C09140=1217.409,7.610,-42.513,-179.514,5.457,148.808
C09141=1217.414,7.361,-42.498,-179.516,5.457,148.808
C09142=1217.419,7.111,-42.484,-179.519,5.456,148.809
C09143=1217.424,6.862,-42.470,-179.521,5.456,148.810
C09144=1217.430,6.611,-42.455,-179.524,5.455,148.810
C09145=1217.434,6.362,-42.440,-179.527,5.455,148.811
C09146=1217.439,6.113,-42.426,-179.529,5.455,148.812
C09147=1217.444,5.863,-42.411,-179.531,5.454,148.812
C09148=1217.450,5.614,-42.397,-179.534,5.454,148.813
C09149=1217.454,5.365,-42.382,-179.537,5.453,148.814
C09150=1217.459,5.115,-42.368,-179.539,5.453,148.814
C09151=1217.464,4.865,-42.354,-179.541,5.453,148.815
C09152=1217.469,4.616,-42.340,-179.544,5.453,148.816
C09153=1217.475,4.366,-42.324,-179.547,5.452,148.817
C09154=1217.480,4.117,-42.310,-179.549,5.452,148.817
C09155=1217.484,3.867,-42.295,-179.552,5.451,148.818
C09156=1217.490,3.598,-42.280,-179.555,5.451,148.819
C09157=1217.496,3.329,-42.265,-179.557,5.450,148.819
C09158=1217.501,3.061,-42.249,-179.559,5.450,148.820
C09159=1217.506,2.791,-42.234,-179.562,5.450,148.821
C09160=1217.511,2.542,-42.219,-179.565,5.449,148.821
C09161=1217.516,2.292,-42.205,-179.567,5.449,148.822
C09162=1217.521,2.043,-42.191,-179.570,5.448,148.823
C09163=1217.526,1.793,-42.176,-179.573,5.448,148.823
C09164=1217.532,1.544,-42.162,-179.575,5.448,148.824
C09165=1217.537,1.294,-42.148,-179.577,5.448,148.825
C09166=1217.542,1.044,-42.134,-179.580,5.447,148.825
C09167=1217.547,0.795,-42.119,-179.583,5.446,148.826
C09168=1217.552,0.545,-42.105,-179.585,5.446,148.827
C09169=1217.557,0.296,-42.091,-179.587,5.446,148.828
C09170=1217.562,0.046,-42.077,-179.589,5.445,148.828
C09171=1217.567,-0.203,-42.062,-179.592,5.445,148.829
C09172=1217.572,-0.453,-42.048,-179.595,5.444,148.829
C09173=1217.577,-0.702,-42.033,-179.597,5.445,148.830
C09174=1217.582,-0.951,-42.019,-179.600,5.444,148.831
C09175=1217.587,-1.201,-42.005,-179.602,5.444,148.831
C09176=1217.592,-1.451,-41.991,-179.605,5.443,148.832
C09177=1217.597,-1.700,-41.977,-179.608,5.443,148.833
C09178=1217.602,-1.950,-41.963,-179.610,5.443,148.833
C09179=1217.607,-2.199,-41.949,-179.612,5.442,148.834
C09180=1217.612,-2.449,-41.935,-179.615,5.442,148.835
C09181=1217.617,-2.698,-41.920,-179.618,5.441,148.836
C09182=1217.622,-2.948,-41.906,-179.620,5.442,148.836
C09183=1217.627,-3.198,-41.892,-179.622,5.441,148.837
C09184=1217.633,-3.447,-41.879,-179.625,5.441,148.838
C09185=1217.638,-3.697,-41.864,-179.628,5.440,148.838
C09186=1217.643,-3.947,-41.850,-179.629,5.440,148.839
C09187=1217.648,-4.197,-41.836,-179.632,5.440,148.839
C09188=1217.653,-4.446,-41.822,-179.634,5.439,148.840
C09189=1217.657,-4.695,-41.808,-179.637,5.439,148.841
C09190=1217.662,-4.945,-41.794,-179.640,5.438,148.842
C09191=1217.667,-5.194,-41.780,-179.642,5.438,148.842
C09192=1217.673,-5.443,-41.766,-179.645,5.438,148.843
C09193=1217.678,-5.693,-41.751,-179.647,5.437,148.844
C09194=1217.683,-5.943,-41.738,-179.650,5.437,148.844
C09195=1217.689,-6.192,-41.724,-179.652,5.437,148.845
C09196=1217.694,-6.442,-41.710,-179.655,5.437,148.846
C09197=1217.698,-6.692,-41.696,-179.657,5.436,148.846
C09198=1217.703,-6.941,-41.682,-179.660,5.436,148.847
C09199=1217.708,-7.190,-41.668,-179.662,5.436,148.848
C09200=1217.713,-7.440,-41.654,-179.665,5.435,148.848
C09201=1217.719,-7.690,-41.640,-179.667,5.435,148.849
C09202=1217.723,-7.939,-41.627,-179.670,5.434,148.850
C09203=1217.728,-8.189,-41.612,-179.672,5.435,148.851
C09204=1217.733,-8.438,-41.598,-179.674,5.434,148.851
C09205=1217.738,-8.688,-41.584,-179.677,5.433,148.852
C09206=1217.744,-8.938,-41.571,-179.679,5.433,148.852
C09207=1217.748,-9.187,-41.557,-179.682,5.433,148.853
C09208=1217.753,-9.437,-41.543,-179.684,5.433,148.854
C09209=1217.759,-9.686,-41.529,-179.687,5.432,148.854
C09210=1217.764,-9.936,-41.515,-179.689,5.432,148.855
C09211=1217.769,-10.186,-41.501,-179.692,5.432,148.856
C09212=1217.774,-10.435,-41.488,-179.694,5.431,148.857
C09213=1217.779,-10.684,-41.473,-179.697,5.431,148.857
C09214=1217.784,-10.935,-41.460,-179.700,5.430,148.858
C09215=1217.790,-11.184,-41.446,-179.702,5.431,148.859
C09216=1217.794,-11.433,-41.432,-179.704,5.430,148.859
C09217=1217.800,-11.683,-41.419,-179.707,5.430,148.860
C09218=1217.805,-11.932,-41.405,-179.710,5.429,148.861
C09219=1217.809,-12.182,-41.391,-179.712,5.430,148.861
C09220=1217.815,-12.431,-41.378,-179.714,5.429,148.862
C09221=1217.820,-12.681,-41.364,-179.717,5.429,148.863
C09222=1217.825,-12.931,-41.349,-179.720,5.428,148.863
C09223=1217.830,-13.180,-41.337,-179.722,5.428,148.864
C09224=1217.835,-13.430,-41.322,-179.724,5.427,148.865
C09225=1217.840,-13.680,-41.308,-179.727,5.427,148.865
C09226=1217.845,-13.929,-41.296,-179.729,5.427,148.866
C09227=1217.850,-14.179,-41.281,-179.731,5.427,148.867
C09228=1217.855,-14.428,-41.267,-179.734,5.426,148.867
C09229=1217.860,-14.678,-41.254,-179.737,5.426,148.868
C09230=1217.865,-14.927,-41.240,-179.739,5.426,148.869
C09231=1217.871,-15.177,-41.227,-179.741,5.426,148.869
C09232=1217.875,-15.426,-41.213,-179.744,5.425,148.870
C09233=1217.881,-15.676,-41.200,-179.747,5.425,148.871
C09234=1217.886,-15.926,-41.186,-179.749,5.425,148.872
C09235=1217.890,-16.174,-41.172,-179.751,5.424,148.872
C09236=1217.896,-16.425,-41.159,-179.754,5.424,148.873
C09237=1217.901,-16.674,-41.145,-179.756,5.424,148.874
C09238=1217.906,-16.924,-41.132,-179.759,5.424,148.874
C09239=1217.911,-17.174,-41.118,-179.761,5.423,148.875
C09240=1217.916,-17.423,-41.105,-179.764,5.423,148.876
C09241=1217.921,-17.673,-41.091,-179.766,5.423,148.876
C09242=1217.927,-17.922,-41.078,-179.769,5.423,148.877
C09243=1217.931,-18.172,-41.064,-179.771,5.422,148.878
C09244=1217.937,-18.421,-41.051,-179.774,5.422,148.878
C09245=1217.941,-18.671,-41.037,-179.776,5.422,148.879
C09246=1217.946,-18.921,-41.023,-179.778,5.421,148.880
C09247=1217.952,-19.170,-41.010,-179.781,5.420,148.880
C09248=1217.956,-19.420,-40.997,-179.783,5.421,148.881
C09249=1217.962,-19.669,-40.983,-179.786,5.420,148.882
C09250=1217.966,-19.919,-40.970,-179.788,5.420,148.882
C09251=1217.972,-20.169,-40.957,-179.791,5.420,148.883
C09252=1217.977,-20.418,-40.943,-179.793,5.420,148.884
C09253=1217.982,-20.668,-40.930,-179.796,5.419,148.884
C09254=1217.987,-20.917,-40.915,-179.798,5.419,148.885
C09255=1217.992,-21.167,-40.903,-179.801,5.419,148.886
C09256=1217.998,-21.417,-40.889,-179.803,5.418,148.887
C09257=1218.003,-21.666,-40.876,-179.806,5.418,148.887
C09258=1218.008,-21.916,-40.862,-179.808,5.418,148.888
C09259=1218.013,-22.165,-40.849,-179.811,5.418,148.889
C09260=1218.018,-22.435,-40.835,-179.813,5.417,148.889
C09261=1218.023,-22.704,-40.820,-179.816,5.417,148.890
C09262=1218.029,-22.973,-40.806,-179.819,5.416,148.891
C09263=1218.035,-23.243,-40.791,-179.821,5.417,148.892
C09264=1218.039,-23.493,-40.778,-179.824,5.417,148.892
C09265=1218.045,-23.742,-40.765,-179.827,5.416,148.893
C09266=1218.049,-23.992,-40.752,-179.829,5.416,148.894
C09267=1218.055,-24.241,-40.738,-179.831,5.416,148.894
C09268=1218.060,-24.491,-40.726,-179.833,5.415,148.895
C09269=1218.065,-24.740,-40.712,-179.836,5.414,148.896
C09270=1218.070,-24.990,-40.699,-179.838,5.415,148.896
C09271=1218.075,-25.240,-40.686,-179.841,5.414,148.897
C09272=1218.081,-25.489,-40.672,-179.843,5.414,148.898
C09273=1218.085,-25.739,-40.659,-179.846,5.414,148.898
C09274=1218.091,-25.988,-40.646,-179.848,5.414,148.899
C09275=1218.095,-26.238,-40.633,-179.851,5.413,148.900
C09276=1218.101,-26.487,-40.619,-179.853,5.413,148.901
C09277=1218.106,-26.737,-40.606,-179.856,5.413,148.901
C09278=1218.111,-26.987,-40.593,-179.858,5.412,148.902
C09279=1218.117,-27.236,-40.580,-179.860,5.413,148.903
C09280=1218.121,-27.486,-40.567,-179.863,5.412,148.903
C09281=1218.127,-27.735,-40.553,-179.866,5.412,148.904
C09282=1218.131,-27.985,-40.540,-179.868,5.411,148.905
C09283=1218.136,-28.235,-40.528,-179.870,5.412,148.905
C09284=1218.142,-28.484,-40.515,-179.873,5.411,148.906
C09285=1218.147,-28.734,-40.502,-179.876,5.411,148.907
C09286=1218.151,-28.983,-40.488,-179.878,5.411,148.907
C09287=1218.157,-29.233,-40.475,-179.880,5.411,148.908
C09288=1218.162,-29.483,-40.462,-179.883,5.410,148.909
C09289=1218.167,-29.732,-40.450,-179.885,5.410,148.910
C09290=1218.172,-29.982,-40.436,-179.888,5.410,148.910
C09291=1218.177,-30.232,-40.423,-179.891,5.409,148.911
C09292=1218.182,-30.482,-40.410,-179.893,5.410,148.912
C09293=1218.187,-30.731,-40.397,-179.895,5.409,148.912
C09294=1218.193,-30.980,-40.384,-179.897,5.408,148.913
C09295=1218.197,-31.230,-40.371,-179.900,5.409,148.914
C09296=1218.203,-31.480,-40.358,-179.902,5.408,148.914
C09297=1218.208,-31.729,-40.345,-179.905,5.408,148.915
C09298=1218.213,-31.979,-40.332,-179.907,5.408,148.916
C09299=1218.218,-32.229,-40.319,-179.910,5.408,148.916
C09300=1218.224,-32.478,-40.306,-179.912,5.407,148.917
C09301=1218.228,-32.728,-40.293,-179.914,5.407,148.918
C09302=1218.233,-32.977,-40.281,-179.917,5.407,148.918
C09303=1218.239,-33.227,-40.268,-179.920,5.406,148.919
C09304=1218.244,-33.477,-40.255,-179.922,5.407,148.920
C09305=1218.249,-33.726,-40.242,-179.924,5.406,148.921
C09306=1218.255,-33.976,-40.229,-179.927,5.406,148.921
C09307=1218.259,-34.226,-40.216,-179.929,5.406,148.922
C09308=1218.264,-34.475,-40.203,-179.932,5.406,148.923
C09309=1218.269,-34.724,-40.191,-179.934,5.405,148.923
C09310=1218.275,-34.975,-40.177,-179.937,5.405,148.924
C09311=1218.280,-35.224,-40.165,-179.939,5.405,148.925
C09312=1218.285,-35.473,-40.152,-179.942,5.404,148.925
C09313=1218.289,-35.723,-40.139,-179.944,5.405,148.926
C09314=1218.295,-35.973,-40.126,-179.947,5.404,148.927
C09315=1218.300,-36.222,-40.113,-179.949,5.404,148.928
C09316=1218.306,-36.472,-40.101,-179.951,5.404,148.928
C09317=1218.310,-36.722,-40.088,-179.954,5.404,148.929
C09318=1218.315,-36.971,-40.075,-179.957,5.403,148.930
C09319=1218.320,-37.220,-40.062,-179.958,5.403,148.930
C09320=1218.326,-37.471,-40.049,-179.961,5.403,148.931
C09321=1218.331,-37.720,-40.036,-179.963,5.403,148.931
C09322=1218.336,-37.969,-40.024,-179.966,5.403,148.932
C09323=1218.341,-38.219,-40.012,-179.968,5.402,148.933
C09324=1218.346,-38.469,-39.999,-179.970,5.402,148.934
C09325=1218.351,-38.719,-39.986,-179.973,5.402,148.934
C09326=1218.357,-38.968,-39.973,-179.976,5.401,148.935
C09327=1218.362,-39.218,-39.960,-179.978,5.402,148.936
C09328=1218.366,-39.468,-39.947,-179.981,5.401,148.936
C09329=1218.371,-39.717,-39.935,-179.983,5.401,148.937
C09330=1218.377,-39.967,-39.923,-179.985,5.401,148.938
C09331=1218.382,-40.216,-39.910,-179.988,5.401,148.938
C09332=1218.387,-40.466,-39.897,-179.991,5.400,148.939
C09333=1218.392,-40.716,-39.884,-179.993,5.400,148.940
C09334=1218.398,-40.965,-39.872,-179.995,5.400,148.941
C09335=1218.403,-41.214,-39.859,-179.997,5.400,148.941
C09336=1218.408,-41.464,-39.847,180.000,5.400,148.942
C09337=1218.413,-41.714,-39.834,179.997,5.399,148.943
C09338=1218.418,-41.964,-39.822,179.995,5.400,148.943
C09339=1218.423,-42.213,-39.809,179.992,5.399,148.944
C09340=1218.428,-42.463,-39.797,179.990,5.399,148.945
C09341=1218.433,-42.713,-39.784,179.988,5.399,148.945
C09342=1218.438,-42.962,-39.771,179.985,5.399,148.946
C09343=1218.443,-43.212,-39.759,179.982,5.398,148.947
C09344=1218.449,-43.462,-39.747,179.981,5.398,148.947
C09345=1218.454,-43.711,-39.734,179.978,5.398,148.948
C09346=1218.458,-43.961,-39.721,179.976,5.398,148.949
C09347=1218.464,-44.211,-39.708,179.973,5.397,148.949
C09348=1218.469,-44.460,-39.696,179.971,5.397,148.950
C09349=1218.475,-44.710,-39.684,179.969,5.397,148.951
C09350=1218.480,-44.959,-39.671,179.966,5.397,148.952
C09351=1218.485,-45.209,-39.659,179.963,5.396,148.952
C09352=1218.490,-45.459,-39.646,179.961,5.397,148.953
C09353=1218.495,-45.708,-39.634,179.959,5.396,148.954
C09354=1218.500,-45.958,-39.622,179.957,5.397,148.954
C09355=1218.505,-46.208,-39.609,179.954,5.396,148.955
C09356=1218.510,-46.457,-39.597,179.951,5.396,148.956
C09357=1218.516,-46.707,-39.585,179.949,5.396,148.956
C09358=1218.521,-46.956,-39.572,179.946,5.395,148.957
C09359=1218.526,-47.206,-39.559,179.944,5.395,148.958
C09360=1218.531,-47.456,-39.547,179.942,5.395,148.959
C09361=1218.536,-47.705,-39.535,179.939,5.395,148.959
C09362=1218.542,-47.955,-39.523,179.937,5.395,148.960
C09363=1218.546,-48.204,-39.511,179.934,5.395,148.961
C09364=1218.552,-48.475,-39.497,179.932,5.394,148.961
C09365=1218.558,-48.744,-39.484,179.929,5.394,148.962
C09366=1218.563,-49.014,-39.471,179.927,5.394,148.963
C09367=1218.568,-49.284,-39.457,179.924,5.394,148.964
C09368=1218.573,-49.534,-39.445,179.922,5.393,148.964
C09369=1218.578,-49.783,-39.433,179.919,5.394,148.965
C09370=1218.584,-50.033,-39.420,179.917,5.393,148.966
C09371=1218.589,-50.283,-39.408,179.915,5.393,148.966
C09372=1218.594,-50.532,-39.396,179.912,5.393,148.967
C09373=1218.600,-50.782,-39.384,179.909,5.392,148.968
C09374=1218.605,-51.031,-39.371,179.907,5.393,148.968
C09375=1218.610,-51.281,-39.359,179.905,5.392,148.969
C09376=1218.615,-51.531,-39.346,179.902,5.392,148.970
C09377=1218.619,-51.781,-39.335,179.900,5.392,148.971
C09378=1218.624,-52.030,-39.322,179.897,5.392,148.971
C09379=1218.630,-52.280,-39.311,179.895,5.392,148.972
C09380=1218.635,-52.529,-39.298,179.892,5.392,148.973
C09381=1218.640,-52.779,-39.286,179.890,5.391,148.973
C09382=1218.646,-53.029,-39.274,179.888,5.391,148.974
C09383=1218.651,-53.279,-39.262,179.885,5.391,148.975
C09384=1218.656,-53.528,-39.250,179.883,5.391,148.975
C09385=1218.661,-53.778,-39.238,179.880,5.391,148.976
C09386=1218.666,-54.027,-39.226,179.878,5.390,148.977
C09387=1218.671,-54.277,-39.213,179.876,5.391,148.978
C09388=1218.677,-54.527,-39.201,179.873,5.390,148.978
C09389=1218.682,-54.776,-39.189,179.871,5.390,148.979
C09390=1218.687,-55.026,-39.177,179.869,5.390,148.979
C09391=1218.692,-55.276,-39.166,179.866,5.389,148.980
C09392=1218.697,-55.526,-39.153,179.864,5.390,148.981
C09393=1218.702,-55.776,-39.141,179.861,5.389,148.982
C09394=1218.707,-56.026,-39.129,179.859,5.390,148.982
C09395=1218.712,-56.275,-39.117,179.856,5.389,148.983
C09396=1218.717,-56.524,-39.105,179.854,5.389,148.984
C09397=1218.722,-56.774,-39.092,179.852,5.389,148.984
C09398=1218.728,-57.024,-39.080,179.849,5.388,148.985
C09399=1218.732,-57.273,-39.069,179.847,5.389,148.986
C09400=1218.738,-57.523,-39.057,179.844,5.388,148.987
C09401=1218.743,-57.773,-39.045,179.842,5.389,148.987
C09402=1218.748,-58.023,-39.033,179.839,5.388,148.988
C09403=1218.753,-58.272,-39.021,179.837,5.388,148.989
C09404=1218.758,-58.521,-39.009,179.835,5.388,148.989
C09405=1218.764,-58.771,-38.997,179.832,5.388,148.990
C09406=1218.769,-59.021,-38.985,179.830,5.388,148.991
C09407=1218.773,-59.270,-38.973,179.827,5.388,148.991
C09408=1218.779,-59.520,-38.961,179.825,5.387,148.992
C09409=1218.784,-59.770,-38.949,179.823,5.387,148.993
C09410=1218.790,-60.019,-38.938,179.820,5.387,148.993
C09411=1218.795,-60.268,-38.926,179.818,5.387,148.994
C09412=1218.800,-60.518,-38.914,179.816,5.386,148.995
C09413=1218.806,-60.768,-38.902,179.813,5.386,148.995
C09414=1218.810,-61.018,-38.891,179.811,5.386,148.996
C09415=1218.815,-61.267,-38.878,179.808,5.386,148.997
C09416=1218.821,-61.517,-38.866,179.806,5.386,148.998
C09417=1218.826,-61.767,-38.855,179.803,5.386,148.998
C09418=1218.831,-62.017,-38.843,179.801,5.386,148.999
C09419=1218.836,-62.267,-38.831,179.799,5.386,149.000
C09420=1218.841,-62.516,-38.819,179.796,5.385,149.000
C09421=1218.846,-62.766,-38.807,179.794,5.385,149.001
C09422=1218.852,-63.016,-38.795,179.791,5.385,149.002
C09423=1218.856,-63.265,-38.784,179.789,5.385,149.002
C09424=1218.862,-63.515,-38.772,179.787,5.385,149.003
C09425=1218.866,-63.765,-38.761,179.784,5.385,149.004
C09426=1218.872,-64.013,-38.749,179.782,5.384,149.004
C09427=1218.878,-64.263,-38.737,179.780,5.384,149.005
C09428=1218.882,-64.513,-38.726,179.778,5.384,149.006
C09429=1218.888,-64.763,-38.714,179.775,5.384,149.007
C09430=1218.893,-65.013,-38.702,179.773,5.384,149.007
C09431=1218.898,-65.262,-38.691,179.770,5.384,149.008
C09432=1218.903,-65.512,-38.679,179.768,5.384,149.009
C09433=1218.908,-65.762,-38.667,179.765,5.384,149.009
C09434=1218.913,-66.012,-38.655,179.763,5.383,149.010
C09435=1218.918,-66.261,-38.643,179.761,5.384,149.011
C09436=1218.924,-66.510,-38.632,179.758,5.383,149.011
C09437=1218.929,-66.760,-38.620,179.756,5.383,149.012
C09438=1218.934,-67.010,-38.609,179.753,5.383,149.013
C09439=1218.939,-67.260,-38.597,179.751,5.383,149.014
C09440=1218.944,-67.509,-38.586,179.748,5.383,149.014
C09441=1218.949,-67.759,-38.574,179.746,5.382,149.015
C09442=1218.954,-68.009,-38.562,179.744,5.382,149.015
C09443=1218.960,-68.258,-38.551,179.741,5.382,149.016
C09444=1218.966,-68.508,-38.539,179.739,5.382,149.017
C09445=1218.970,-68.758,-38.528,179.737,5.382,149.018
C09446=1218.976,-69.008,-38.516,179.735,5.382,149.018
C09447=1218.980,-69.257,-38.505,179.732,5.382,149.019
C09448=1218.986,-69.507,-38.493,179.730,5.382,149.020
C09449=1218.991,-69.756,-38.482,179.727,5.382,149.020
C09450=1218.997,-70.006,-38.470,179.724,5.381,149.021
C09451=1219.001,-70.256,-38.459,179.722,5.381,149.022
C09452=1219.007,-70.506,-38.447,179.720,5.381,149.023
C09453=1219.011,-70.755,-38.435,179.718,5.381,149.023
C09454=1219.017,-71.005,-38.423,179.715,5.381,149.024
C09455=1219.022,-71.254,-38.413,179.713,5.381,149.025
C09456=1219.028,-71.504,-38.401,179.710,5.381,149.025
C09457=1219.033,-71.754,-38.390,179.709,5.381,149.026
C09458=1219.038,-72.004,-38.378,179.706,5.380,149.027
C09459=1219.043,-72.254,-38.367,179.703,5.380,149.027
C09460=1219.049,-72.503,-38.355,179.701,5.380,149.028
C09461=1219.053,-72.753,-38.344,179.699,5.380,149.029
C09462=1219.058,-73.002,-38.333,179.696,5.380,149.029
C09463=1219.064,-73.252,-38.321,179.694,5.380,149.030
C09464=1219.069,-73.501,-38.310,179.692,5.380,149.031
C09465=1219.074,-73.751,-38.298,179.689,5.380,149.032
C09466=1219.079,-74.001,-38.288,179.687,5.380,149.032
C09467=1219.085,-74.251,-38.276,179.684,5.379,149.033
C09468=1219.091,-74.521,-38.263,179.682,5.379,149.034
C09469=1219.095,-74.792,-38.251,179.680,5.379,149.034
C09470=1219.101,-75.063,-38.239,179.677,5.379,149.035
C09471=1219.107,-75.332,-38.227,179.674,5.379,149.036
C09472=1219.112,-75.583,-38.216,179.672,5.379,149.036
C09473=1219.117,-75.832,-38.204,179.669,5.378,149.037
C09474=1219.122,-76.082,-38.193,179.667,5.379,149.038
C09475=1219.128,-76.331,-38.181,179.665,5.378,149.039
C09476=1219.133,-76.581,-38.170,179.663,5.379,149.039
C09477=1219.138,-76.831,-38.159,179.660,5.378,149.040
C09478=1219.144,-77.080,-38.148,179.658,5.379,149.041
C09479=1219.149,-77.330,-38.137,179.655,5.378,149.041
C09480=1219.154,-77.580,-38.125,179.652,5.378,149.042
C09481=1219.159,-77.830,-38.114,179.650,5.378,149.043
C09482=1219.164,-78.079,-38.103,179.648,5.377,149.043
C09483=1219.170,-78.329,-38.091,179.646,5.378,149.044
C09484=1219.174,-78.579,-38.080,179.643,5.377,149.045
C09485=1219.179,-78.829,-38.069,179.641,5.377,149.045
C09486=1219.185,-79.078,-38.058,179.639,5.377,149.046
C09487=1219.190,-79.328,-38.047,179.637,5.377,149.047
C09488=1219.195,-79.578,-38.036,179.634,5.377,149.048
C09489=1219.200,-79.827,-38.025,179.632,5.377,149.048
C09490=1219.206,-80.077,-38.013,179.629,5.377,149.049
C09491=1219.211,-80.327,-38.002,179.627,5.377,149.050
C09492=1219.216,-80.576,-37.992,179.624,5.377,149.050
C09493=1219.222,-80.826,-37.980,179.622,5.377,149.051
C09494=1219.226,-81.076,-37.969,179.620,5.376,149.052
C09495=1219.232,-81.325,-37.958,179.617,5.376,149.052
C09496=1219.237,-81.575,-37.947,179.615,5.376,149.053
C09497=1219.242,-81.825,-37.936,179.613,5.376,149.054
C09498=1219.248,-82.074,-37.925,179.611,5.376,149.054
C09499=1219.252,-82.324,-37.914,179.608,5.376,149.055
C09500=1219.258,-82.574,-37.903,179.606,5.376,149.056
C09501=1219.263,-82.823,-37.892,179.603,5.376,149.057
C09502=1219.268,-83.073,-37.880,179.601,5.376,149.057
C09503=1219.273,-83.323,-37.870,179.598,5.376,149.058
C09504=1219.278,-83.572,-37.859,179.596,5.376,149.059
C09505=1219.284,-83.823,-37.848,179.594,5.375,149.059
C09506=1219.289,-84.072,-37.836,179.592,5.375,149.060
C09507=1219.294,-84.321,-37.825,179.589,5.375,149.061
C09508=1219.299,-84.572,-37.815,179.587,5.375,149.061
C09509=1219.304,-84.821,-37.803,179.585,5.375,149.062
C09510=1219.310,-85.071,-37.793,179.583,5.375,149.063
C09511=1219.315,-85.321,-37.782,179.580,5.375,149.063
C09512=1219.320,-85.570,-37.771,179.578,5.375,149.064
C09513=1219.325,-85.820,-37.760,179.575,5.375,149.065
C09514=1219.331,-86.070,-37.749,179.572,5.374,149.066
C09515=1219.336,-86.319,-37.738,179.571,5.374,149.066
C09516=1219.341,-86.570,-37.727,179.568,5.374,149.067
C09517=1219.346,-86.819,-37.716,179.566,5.374,149.067
C09518=1219.351,-87.069,-37.706,179.563,5.374,149.068
C09519=1219.356,-87.318,-37.695,179.561,5.374,149.069
C09520=1219.362,-87.568,-37.684,179.559,5.374,149.070
C09521=1219.367,-87.818,-37.672,179.557,5.374,149.070
C09522=1219.372,-88.068,-37.662,179.554,5.374,149.071
C09523=1219.377,-88.317,-37.651,179.552,5.374,149.072
C09524=1219.382,-88.567,-37.640,179.549,5.373,149.072
C09525=1219.388,-88.816,-37.629,179.547,5.373,149.073
C09526=1219.393,-89.066,-37.619,179.545,5.373,149.074
C09527=1219.398,-89.315,-37.608,179.543,5.373,149.074
C09528=1219.404,-89.566,-37.597,179.540,5.373,149.075
C09529=1219.409,-89.816,-37.586,179.538,5.373,149.076
C09530=1219.414,-90.065,-37.575,179.535,5.373,149.076
C09531=1219.419,-90.315,-37.565,179.533,5.373,149.077
C09532=1219.424,-90.564,-37.554,179.531,5.373,149.078
C09533=1219.429,-90.814,-37.543,179.528,5.373,149.079
C09534=1219.435,-91.064,-37.533,179.526,5.372,149.079
C09535=1219.440,-91.314,-37.522,179.524,5.373,149.080
C09536=1219.445,-91.563,-37.512,179.521,5.372,149.081
C09537=1219.450,-91.813,-37.501,179.519,5.373,149.081
C09538=1219.455,-92.062,-37.490,179.517,5.372,149.082
C09539=1219.460,-92.313,-37.479,179.515,5.373,149.083
C09540=1219.466,-92.563,-37.468,179.512,5.372,149.083
C09541=1219.471,-92.812,-37.457,179.510,5.373,149.084
C09542=1219.476,-93.062,-37.447,179.508,5.372,149.085
C09543=1219.482,-93.311,-37.436,179.506,5.372,149.085
C09544=1219.487,-93.561,-37.425,179.503,5.372,149.086
C09545=1219.492,-93.811,-37.415,179.501,5.372,149.087
C09546=1219.497,-94.061,-37.404,179.498,5.372,149.087
C09547=1219.503,-94.310,-37.394,179.496,5.372,149.088
C09548=1219.508,-94.560,-37.383,179.493,5.371,149.089
C09549=1219.513,-94.810,-37.373,179.491,5.372,149.090
C09550=1219.518,-95.060,-37.361,179.489,5.371,149.090
C09551=1219.523,-95.309,-37.351,179.487,5.371,149.091
C09552=1219.528,-95.559,-37.341,179.484,5.371,149.091
C09553=1219.534,-95.809,-37.330,179.482,5.371,149.092
C09554=1219.539,-96.059,-37.319,179.480,5.371,149.093
C09555=1219.544,-96.308,-37.309,179.477,5.371,149.094
C09556=1219.550,-96.558,-37.299,179.475,5.371,149.094
C09557=1219.555,-96.808,-37.288,179.473,5.371,149.095
C09558=1219.560,-97.057,-37.277,179.471,5.370,149.096
C09559=1219.565,-97.307,-37.267,179.468,5.371,149.096
C09560=1219.571,-97.557,-37.257,179.466,5.370,149.097
C09561=1219.576,-97.807,-37.246,179.464,5.371,149.098
C09562=1219.581,-98.056,-37.236,179.461,5.370,149.098
C09563=1219.586,-98.306,-37.224,179.459,5.371,149.099
C09564=1219.591,-98.555,-37.215,179.456,5.370,149.100
C09565=1219.596,-98.806,-37.204,179.454,5.371,149.100
C09566=1219.602,-99.055,-37.194,179.452,5.370,149.101
C09567=1219.607,-99.305,-37.184,179.450,5.370,149.102
C09568=1219.612,-99.555,-37.173,179.447,5.370,149.102
C09569=1219.617,-99.804,-37.162,179.445,5.370,149.103
C09570=1219.622,-100.054,-37.152,179.442,5.370,149.104
C09571=1219.628,-100.304,-37.142,179.440,5.370,149.105
C09572=1219.633,-100.575,-37.131,179.438,5.370,149.105
C09573=1219.639,-100.846,-37.119,179.435,5.369,149.106
C09574=1219.645,-101.117,-37.108,179.433,5.370,149.107
C09575=1219.651,-101.388,-37.096,179.430,5.369,149.107
C09576=1219.656,-101.638,-37.086,179.428,5.369,149.108
C09577=1219.661,-101.888,-37.075,179.425,5.369,149.109
C09578=1219.666,-102.137,-37.066,179.423,5.369,149.110
C09579=1219.671,-102.387,-37.055,179.421,5.369,149.110
C09580=1219.677,-102.637,-37.045,179.419,5.369,149.111
C09581=1219.682,-102.886,-37.035,179.416,5.369,149.111
C09582=1219.687,-103.137,-37.024,179.414,5.369,149.112
C09583=1219.693,-103.386,-37.014,179.412,5.368,149.113
C09584=1219.698,-103.636,-37.003,179.410,5.369,149.114
C09585=1219.703,-103.886,-36.994,179.407,5.368,149.114
C09586=1219.708,-104.135,-36.984,179.405,5.369,149.115
C09587=1219.713,-104.385,-36.973,179.403,5.368,149.116
C09588=1219.719,-104.635,-36.963,179.401,5.368,149.116
C09589=1219.724,-104.885,-36.953,179.398,5.368,149.117
C09590=1219.729,-105.134,-36.943,179.396,5.368,149.118
C09591=1219.734,-105.384,-36.932,179.393,5.368,149.118
C09592=1219.739,-105.634,-36.922,179.391,5.368,149.119
C09593=1219.745,-105.884,-36.912,179.389,5.368,149.120
C09594=1219.751,-106.133,-36.902,179.387,5.368,149.120
C09595=1219.755,-106.383,-36.892,179.385,5.368,149.121
C09596=1219.760,-106.633,-36.881,179.382,5.368,149.122
C09597=1219.766,-106.882,-36.871,179.380,5.368,149.122
C09598=1219.771,-107.133,-36.861,179.377,5.368,149.123
C09599=1219.776,-107.382,-36.851,179.375,5.368,149.124
C09600=1219.781,-107.631,-36.841,179.373,5.367,149.124
C09601=1219.786,-107.882,-36.830,179.371,5.368,149.125
C09602=1219.792,-108.131,-36.820,179.368,5.367,149.126
C09603=1219.798,-108.381,-36.810,179.366,5.368,149.126
C09604=1219.802,-108.631,-36.800,179.363,5.367,149.127
C09605=1219.808,-108.880,-36.790,179.361,5.368,149.128
C09606=1219.813,-109.130,-36.779,179.359,5.367,149.128
C09607=1219.818,-109.380,-36.770,179.357,5.367,149.129
C09608=1219.823,-109.630,-36.760,179.354,5.367,149.130
C09609=1219.829,-109.879,-36.750,179.352,5.367,149.131
C09610=1219.834,-110.129,-36.739,179.350,5.367,149.131
C09611=1219.839,-110.379,-36.729,179.347,5.367,149.132
C09612=1219.844,-110.628,-36.719,179.345,5.366,149.132
C09613=1219.850,-110.878,-36.709,179.343,5.367,149.133
C09614=1219.854,-111.128,-36.699,179.341,5.367,149.134
C09615=1219.860,-111.378,-36.690,179.338,5.367,149.135
C09616=1219.866,-111.628,-36.679,179.336,5.367,149.135
C09617=1219.871,-111.877,-36.670,179.334,5.366,149.136
C09618=1219.876,-112.127,-36.659,179.332,5.367,149.136
C09619=1219.881,-112.377,-36.649,179.329,5.366,149.137
C09620=1219.886,-112.626,-36.640,179.327,5.366,149.138
C09621=1219.892,-112.876,-36.630,179.325,5.366,149.139
C09622=1219.897,-113.126,-36.619,179.322,5.366,149.139
C09623=1219.902,-113.375,-36.610,179.320,5.366,149.140
C09624=1219.907,-113.625,-36.599,179.318,5.366,149.141
C09625=1219.913,-113.875,-36.590,179.316,5.366,149.141
C09626=1219.918,-114.125,-36.580,179.313,5.366,149.142
C09627=1219.923,-114.375,-36.570,179.311,5.366,149.143
C09628=1219.929,-114.624,-36.560,179.309,5.366,149.143
C09629=1219.934,-114.874,-36.551,179.307,5.366,149.144
C09630=1219.939,-115.124,-36.540,179.304,5.366,149.145
C09631=1219.944,-115.374,-36.530,179.302,5.366,149.145
C09632=1219.949,-115.623,-36.520,179.300,5.365,149.146
C09633=1219.955,-115.873,-36.511,179.298,5.365,149.147
C09634=1219.960,-116.122,-36.501,179.295,5.365,149.147
C09635=1219.965,-116.373,-36.491,179.293,5.365,149.148
C09636=1219.971,-116.623,-36.481,179.291,5.365,149.149
C09637=1219.976,-116.872,-36.471,179.288,5.365,149.149
C09638=1219.981,-117.122,-36.461,179.286,5.365,149.150
C09639=1219.987,-117.371,-36.452,179.284,5.365,149.151
C09640=1219.992,-117.622,-36.442,179.281,5.365,149.151
C09641=1219.997,-117.871,-36.432,179.279,5.365,149.152
C09642=1220.002,-118.121,-36.423,179.277,5.365,149.153
C09643=1220.008,-118.371,-36.412,179.275,5.365,149.153
C09644=1220.013,-118.620,-36.403,179.273,5.365,149.154
C09645=1220.018,-118.871,-36.393,179.270,5.364,149.155
C09646=1220.023,-119.120,-36.383,179.268,5.365,149.155
C09647=1220.029,-119.370,-36.373,179.266,5.364,149.156
C09648=1220.034,-119.619,-36.364,179.264,5.364,149.157
C09649=1220.039,-119.869,-36.354,179.261,5.364,149.157
C09650=1220.044,-120.119,-36.345,179.259,5.364,149.158
C09651=1220.050,-120.369,-36.335,179.257,5.364,149.159
C09652=1220.054,-120.618,-36.325,179.254,5.364,149.159
C09653=1220.060,-120.868,-36.316,179.252,5.364,149.160
C09654=1220.065,-121.118,-36.306,179.250,5.364,149.161
C09655=1220.071,-121.368,-36.296,179.248,5.364,149.161
C09656=1220.076,-121.617,-36.287,179.245,5.364,149.162
C09657=1220.081,-121.868,-36.277,179.243,5.364,149.163
C09658=1220.086,-122.117,-36.267,179.241,5.364,149.163
C09659=1220.092,-122.367,-36.257,179.239,5.364,149.164
C09660=1220.097,-122.617,-36.248,179.236,5.363,149.165
C09661=1220.102,-122.866,-36.238,179.234,5.364,149.165
C09662=1220.108,-123.116,-36.229,179.232,5.363,149.166
C09663=1220.113,-123.365,-36.219,179.230,5.363,149.167
C09664=1220.118,-123.616,-36.210,179.227,5.363,149.167
C09665=1220.123,-123.865,-36.200,179.225,5.363,149.168
C09666=1220.129,-124.115,-36.191,179.223,5.364,149.169
C09667=1220.133,-124.365,-36.181,179.221,5.363,149.169
C09668=1220.139,-124.615,-36.171,179.219,5.363,149.170
C09669=1220.144,-124.864,-36.162,179.216,5.363,149.171
C09670=1220.150,-125.114,-36.152,179.214,5.363,149.171
C09671=1220.155,-125.363,-36.143,179.212,5.363,149.172
C09672=1220.160,-125.613,-36.134,179.210,5.363,149.173
C09673=1220.166,-125.863,-36.124,179.207,5.363,149.173
C09674=1220.170,-126.113,-36.114,179.205,5.363,149.174
C09675=1220.176,-126.364,-36.105,179.202,5.363,149.175
C09676=1219.755,-126.374,-36.142,179.198,5.366,149.177
C09677=1219.749,-126.123,-36.151,179.201,5.366,149.176
C09678=1219.744,-125.874,-36.161,179.203,5.366,149.175
C09679=1219.738,-125.624,-36.170,179.205,5.367,149.175
C09680=1219.734,-125.375,-36.180,179.207,5.366,149.174
C09681=1219.728,-125.125,-36.189,179.210,5.367,149.173
C09682=1219.723,-124.875,-36.199,179.212,5.366,149.173
C09683=1219.718,-124.626,-36.208,179.214,5.367,149.172
C09684=1219.712,-124.375,-36.217,179.216,5.367,149.171
C09685=1219.707,-124.126,-36.227,179.219,5.367,149.171
C09686=1219.702,-123.875,-36.237,179.221,5.367,149.170
C09687=1219.697,-123.626,-36.246,179.223,5.367,149.169
C09688=1219.691,-123.376,-36.255,179.226,5.367,149.169
C09689=1219.686,-123.127,-36.265,179.228,5.367,149.168
C09690=1219.681,-122.877,-36.275,179.230,5.367,149.167
C09691=1219.675,-122.627,-36.285,179.232,5.367,149.167
C09692=1219.670,-122.378,-36.294,179.235,5.367,149.166
C09693=1219.664,-122.128,-36.304,179.237,5.367,149.165
C09694=1219.660,-121.878,-36.314,179.239,5.367,149.165
C09695=1219.654,-121.628,-36.323,179.241,5.367,149.164
C09696=1219.649,-121.379,-36.333,179.244,5.368,149.163
C09697=1219.643,-121.128,-36.342,179.246,5.368,149.163
C09698=1219.639,-120.879,-36.352,179.248,5.367,149.162
C09699=1219.633,-120.629,-36.361,179.250,5.368,149.161
C09700=1219.628,-120.380,-36.371,179.253,5.367,149.161
C09701=1219.623,-120.130,-36.382,179.255,5.368,149.160
C09702=1219.618,-119.880,-36.390,179.257,5.368,149.159
C09703=1219.612,-119.630,-36.401,179.260,5.368,149.159
C09704=1219.607,-119.380,-36.410,179.262,5.368,149.158
C09705=1219.601,-119.131,-36.420,179.264,5.368,149.157
C09706=1219.596,-118.882,-36.429,179.266,5.368,149.157
C09707=1219.591,-118.631,-36.439,179.269,5.368,149.156
C09708=1219.586,-118.381,-36.449,179.271,5.368,149.155
C09709=1219.581,-118.132,-36.459,179.273,5.368,149.155
C09710=1219.575,-117.882,-36.468,179.275,5.368,149.154
C09711=1219.570,-117.632,-36.478,179.277,5.368,149.153
C09712=1219.565,-117.382,-36.489,179.280,5.369,149.153
C09713=1219.560,-117.132,-36.498,179.282,5.368,149.152
C09714=1219.554,-116.883,-36.508,179.285,5.369,149.151
C09715=1219.549,-116.634,-36.517,179.286,5.369,149.151
C09716=1219.543,-116.383,-36.527,179.289,5.369,149.150
C09717=1219.539,-116.133,-36.537,179.291,5.369,149.149
C09718=1219.533,-115.884,-36.547,179.294,5.369,149.149
C09719=1219.528,-115.634,-36.557,179.296,5.369,149.148
C09720=1219.523,-115.385,-36.566,179.298,5.369,149.147
C09721=1219.518,-115.134,-36.577,179.300,5.369,149.147
C09722=1219.512,-114.885,-36.587,179.302,5.369,149.146
C09723=1219.507,-114.635,-36.596,179.305,5.369,149.145
C09724=1219.501,-114.385,-36.606,179.307,5.369,149.145
C09725=1219.497,-114.136,-36.616,179.309,5.369,149.144
C09726=1219.492,-113.886,-36.626,179.311,5.369,149.143
C09727=1219.486,-113.636,-36.636,179.314,5.370,149.143
C09728=1219.481,-113.387,-36.645,179.316,5.369,149.142
C09729=1219.475,-113.137,-36.656,179.319,5.370,149.141
C09730=1219.470,-112.887,-36.666,179.321,5.369,149.141
C09731=1219.465,-112.637,-36.675,179.323,5.370,149.140
C09732=1219.459,-112.387,-36.685,179.325,5.370,149.139
C09733=1219.454,-112.138,-36.696,179.328,5.370,149.139
C09734=1219.450,-111.888,-36.706,179.330,5.370,149.138
C09735=1219.444,-111.638,-36.716,179.332,5.370,149.137
C09736=1219.438,-111.389,-36.726,179.334,5.370,149.137
C09737=1219.433,-111.139,-36.735,179.337,5.371,149.136
C09738=1219.428,-110.889,-36.745,179.339,5.370,149.135
C09739=1219.423,-110.639,-36.756,179.341,5.370,149.135
C09740=1219.418,-110.390,-36.765,179.343,5.370,149.134
C09741=1219.413,-110.140,-36.776,179.346,5.370,149.133
C09742=1219.407,-109.890,-36.786,179.348,5.371,149.133
C09743=1219.401,-109.640,-36.795,179.350,5.370,149.132
C09744=1219.397,-109.390,-36.805,179.353,5.371,149.131
C09745=1219.391,-109.140,-36.816,179.355,5.370,149.130
C09746=1219.386,-108.891,-36.826,179.357,5.371,149.130
C09747=1219.381,-108.642,-36.836,179.359,5.370,149.129
C09748=1219.376,-108.391,-36.846,179.362,5.371,149.129
C09749=1219.370,-108.142,-36.856,179.364,5.371,149.128
C09750=1219.365,-107.892,-36.866,179.366,5.371,149.127
C09751=1219.360,-107.642,-36.876,179.368,5.371,149.126
C09752=1219.355,-107.393,-36.887,179.371,5.371,149.126
C09753=1219.349,-107.143,-36.897,179.373,5.371,149.125
C09754=1219.344,-106.892,-36.907,179.375,5.372,149.125
C09755=1219.339,-106.643,-36.916,179.377,5.371,149.124
C09756=1219.333,-106.394,-36.927,179.380,5.372,149.123
C09757=1219.328,-106.143,-36.937,179.382,5.371,149.122
C09758=1219.323,-105.894,-36.947,179.385,5.372,149.122
C09759=1219.317,-105.644,-36.958,179.387,5.371,149.121
C09760=1219.313,-105.394,-36.968,179.389,5.371,149.120
C09761=1219.307,-105.145,-36.978,179.391,5.372,149.120
C09762=1219.302,-104.895,-36.988,179.393,5.371,149.119
C09763=1219.297,-104.645,-36.999,179.396,5.372,149.118
C09764=1219.291,-104.396,-37.009,179.398,5.372,149.118
C09765=1219.287,-104.146,-37.019,179.401,5.372,149.117
C09766=1219.281,-103.896,-37.029,179.402,5.372,149.116
C09767=1219.276,-103.647,-37.039,179.405,5.372,149.116
C09768=1219.271,-103.396,-37.050,179.407,5.372,149.115
C09769=1219.265,-103.147,-37.060,179.410,5.372,149.114
C09770=1219.260,-102.898,-37.071,179.412,5.372,149.114
C09771=1219.256,-102.648,-37.081,179.415,5.372,149.113
C09772=1219.250,-102.398,-37.091,179.417,5.372,149.112
C09773=1219.245,-102.148,-37.102,179.419,5.373,149.112
C09774=1219.239,-101.899,-37.112,179.421,5.373,149.111
C09775=1219.234,-101.649,-37.122,179.424,5.373,149.110
C09776=1219.229,-101.399,-37.133,179.426,5.373,149.110
C09777=1219.224,-101.127,-37.144,179.428,5.373,149.109
C09778=1219.217,-100.857,-37.155,179.431,5.373,149.108
C09779=1219.212,-100.586,-37.166,179.433,5.373,149.107
C09780=1219.206,-100.314,-37.178,179.436,5.374,149.107
C09781=1219.201,-100.065,-37.188,179.438,5.373,149.106
C09782=1219.196,-99.815,-37.198,179.441,5.374,149.105
C09783=1219.191,-99.565,-37.208,179.443,5.373,149.105
C09784=1219.185,-99.316,-37.219,179.445,5.374,149.104
C09785=1219.180,-99.065,-37.229,179.448,5.373,149.103
C09786=1219.175,-98.817,-37.240,179.450,5.374,149.102
C09787=1219.170,-98.566,-37.251,179.452,5.374,149.102
C09788=1219.164,-98.317,-37.261,179.454,5.374,149.101
C09789=1219.159,-98.067,-37.271,179.457,5.374,149.100
C09790=1219.154,-97.817,-37.282,179.459,5.374,149.100
C09791=1219.149,-97.567,-37.292,179.461,5.374,149.099
C09792=1219.143,-97.318,-37.303,179.464,5.374,149.098
C09793=1219.138,-97.068,-37.313,179.466,5.374,149.098
C09794=1219.133,-96.818,-37.324,179.468,5.375,149.097
C09795=1219.127,-96.568,-37.334,179.470,5.374,149.096
C09796=1219.123,-96.319,-37.345,179.473,5.375,149.096
C09797=1219.117,-96.069,-37.356,179.475,5.374,149.095
C09798=1219.112,-95.819,-37.366,179.478,5.375,149.094
C09799=1219.106,-95.570,-37.376,179.480,5.374,149.094
C09800=1219.102,-95.320,-37.388,179.483,5.375,149.093
C09801=1219.096,-95.070,-37.398,179.485,5.375,149.092
C09802=1219.091,-94.820,-37.408,179.487,5.375,149.092
C09803=1219.086,-94.571,-37.419,179.489,5.375,149.091
C09804=1219.081,-94.321,-37.430,179.492,5.375,149.090
C09805=1219.075,-94.071,-37.440,179.494,5.375,149.090
C09806=1219.070,-93.821,-37.451,179.496,5.375,149.089
C09807=1219.065,-93.572,-37.462,179.498,5.375,149.088
C09808=1219.060,-93.322,-37.472,179.501,5.376,149.087
C09809=1219.054,-93.072,-37.482,179.503,5.375,149.087
C09810=1219.049,-92.822,-37.493,179.505,5.376,149.086
C09811=1219.044,-92.573,-37.504,179.507,5.376,149.085
C09812=1219.039,-92.323,-37.514,179.510,5.376,149.085
C09813=1219.033,-92.073,-37.525,179.512,5.376,149.084
C09814=1219.029,-91.824,-37.536,179.515,5.376,149.083
C09815=1219.023,-91.574,-37.546,179.517,5.376,149.083
C09816=1219.018,-91.325,-37.557,179.520,5.376,149.082
C09817=1219.013,-91.075,-37.568,179.522,5.376,149.081
C09818=1219.008,-90.825,-37.578,179.524,5.376,149.080
C09819=1219.003,-90.575,-37.590,179.526,5.376,149.080
C09820=1218.997,-90.325,-37.600,179.529,5.377,149.079
C09821=1218.992,-90.075,-37.611,179.531,5.376,149.079
C09822=1218.987,-89.826,-37.622,179.534,5.377,149.078
C09823=1218.982,-89.576,-37.632,179.536,5.376,149.077
C09824=1218.976,-89.327,-37.643,179.538,5.377,149.076
C09825=1218.971,-89.077,-37.654,179.540,5.377,149.076
C09826=1218.966,-88.828,-37.665,179.543,5.377,149.075
C09827=1218.961,-88.578,-37.675,179.545,5.377,149.075
C09828=1218.956,-88.327,-37.686,179.547,5.377,149.074
C09829=1218.950,-88.078,-37.698,179.549,5.377,149.073
C09830=1218.945,-87.828,-37.708,179.552,5.378,149.072
C09831=1218.940,-87.579,-37.719,179.554,5.377,149.072
C09832=1218.935,-87.329,-37.730,179.557,5.378,149.071
C09833=1218.930,-87.079,-37.741,179.559,5.377,149.070
C09834=1218.924,-86.830,-37.751,179.562,5.378,149.070
C09835=1218.920,-86.580,-37.762,179.564,5.378,149.069
C09836=1218.913,-86.330,-37.773,179.566,5.378,149.068
C09837=1218.909,-86.081,-37.784,179.569,5.379,149.068
C09838=1218.904,-85.830,-37.795,179.571,5.378,149.067
C09839=1218.898,-85.581,-37.806,179.573,5.379,149.066
C09840=1218.893,-85.331,-37.817,179.575,5.378,149.066
C09841=1218.887,-85.082,-37.828,179.578,5.379,149.065
C09842=1218.882,-84.832,-37.839,179.580,5.378,149.064
C09843=1218.878,-84.582,-37.850,179.583,5.379,149.063
C09844=1218.872,-84.333,-37.861,179.585,5.378,149.063
C09845=1218.867,-84.083,-37.871,179.588,5.379,149.062
C09846=1218.862,-83.833,-37.883,179.590,5.379,149.061
C09847=1218.856,-83.583,-37.894,179.592,5.379,149.061
C09848=1218.852,-83.334,-37.905,179.594,5.379,149.060
C09849=1218.847,-83.083,-37.915,179.597,5.379,149.059
C09850=1218.841,-82.835,-37.926,179.599,5.379,149.059
C09851=1218.836,-82.585,-37.938,179.601,5.380,149.058
C09852=1218.831,-82.334,-37.949,179.603,5.379,149.057
C09853=1218.826,-82.085,-37.960,179.606,5.380,149.057
C09854=1218.821,-81.836,-37.971,179.608,5.379,149.056
C09855=1218.815,-81.585,-37.982,179.611,5.380,149.055
C09856=1218.810,-81.336,-37.993,179.614,5.380,149.054
C09857=1218.805,-81.086,-38.004,179.615,5.380,149.054
C09858=1218.799,-80.836,-38.016,179.618,5.381,149.053
C09859=1218.794,-80.587,-38.026,179.620,5.380,149.053
C09860=1218.789,-80.337,-38.037,179.623,5.381,149.052
C09861=1218.785,-80.087,-38.048,179.625,5.380,149.051
C09862=1218.778,-79.838,-38.060,179.627,5.381,149.050
C09863=1218.774,-79.588,-38.071,179.629,5.380,149.050
C09864=1218.769,-79.338,-38.082,179.632,5.381,149.049
C09865=1218.763,-79.089,-38.093,179.634,5.380,149.048
C09866=1218.758,-78.839,-38.105,179.637,5.381,149.048
C09867=1218.753,-78.589,-38.115,179.639,5.381,149.047
C09868=1218.747,-78.340,-38.127,179.641,5.381,149.046
C09869=1218.742,-78.090,-38.138,179.644,5.382,149.046
C09870=1218.738,-77.841,-38.149,179.646,5.382,149.045
C09871=1218.732,-77.590,-38.160,179.649,5.382,149.044
C09872=1218.727,-77.341,-38.171,179.651,5.382,149.044
C09873=1218.722,-77.092,-38.183,179.653,5.382,149.043
C09874=1218.717,-76.842,-38.194,179.655,5.382,149.042
C09875=1218.712,-76.591,-38.205,179.658,5.382,149.041
C09876=1218.706,-76.342,-38.216,179.660,5.382,149.041
C09877=1218.701,-76.093,-38.228,179.663,5.382,149.040
C09878=1218.696,-75.843,-38.239,179.665,5.382,149.039
C09879=1218.690,-75.593,-38.250,179.668,5.382,149.039
C09880=1218.685,-75.343,-38.261,179.669,5.382,149.038
C09881=1218.680,-75.073,-38.274,179.672,5.382,149.037
C09882=1218.674,-74.803,-38.286,179.675,5.383,149.036
C09883=1218.668,-74.532,-38.298,179.677,5.383,149.036
C09884=1218.663,-74.262,-38.311,179.680,5.383,149.035
C09885=1218.658,-74.011,-38.322,179.682,5.383,149.034
C09886=1218.652,-73.762,-38.333,179.685,5.383,149.034
C09887=1218.647,-73.512,-38.345,179.687,5.384,149.033
C09888=1218.642,-73.263,-38.356,179.689,5.383,149.032
C09889=1218.637,-73.013,-38.368,179.692,5.384,149.031
C09890=1218.631,-72.764,-38.379,179.694,5.383,149.031
C09891=1218.626,-72.514,-38.391,179.697,5.384,149.030
C09892=1218.621,-72.264,-38.402,179.699,5.384,149.029
C09893=1218.616,-72.014,-38.413,179.701,5.384,149.029
C09894=1218.611,-71.764,-38.424,179.704,5.385,149.028
C09895=1218.606,-71.515,-38.435,179.706,5.384,149.027
C09896=1218.600,-71.265,-38.447,179.708,5.385,149.027
C09897=1218.596,-71.016,-38.459,179.711,5.384,149.026
C09898=1218.590,-70.766,-38.470,179.713,5.385,149.025
C09899=1218.585,-70.516,-38.482,179.715,5.384,149.025
C09900=1218.579,-70.267,-38.493,179.718,5.385,149.024
C09901=1218.575,-70.017,-38.505,179.721,5.385,149.023
C09902=1218.569,-69.767,-38.516,179.723,5.385,149.023
C09903=1218.565,-69.518,-38.528,179.725,5.386,149.022
C09904=1218.559,-69.268,-38.540,179.727,5.385,149.021
C09905=1218.554,-69.019,-38.550,179.730,5.386,149.020
C09906=1218.548,-68.769,-38.562,179.732,5.386,149.020
C09907=1218.544,-68.519,-38.574,179.734,5.386,149.019
C09908=1218.538,-68.269,-38.586,179.736,5.386,149.019
C09909=1218.533,-68.019,-38.597,179.739,5.386,149.018
C09910=1218.528,-67.770,-38.609,179.742,5.387,149.017
C09911=1218.523,-67.520,-38.621,179.744,5.386,149.016
C09912=1218.517,-67.271,-38.632,179.747,5.387,149.016
C09913=1218.512,-67.021,-38.643,179.749,5.386,149.015
C09914=1218.507,-66.771,-38.655,179.751,5.387,149.014
C09915=1218.502,-66.521,-38.667,179.753,5.387,149.014
C09916=1218.497,-66.272,-38.678,179.756,5.387,149.013
C09917=1218.492,-66.022,-38.690,179.759,5.387,149.012
C09918=1218.486,-65.772,-38.702,179.761,5.387,149.011
C09919=1218.482,-65.522,-38.713,179.764,5.388,149.011
C09920=1218.476,-65.273,-38.724,179.766,5.387,149.010
C09921=1218.471,-65.024,-38.736,179.768,5.388,149.010
C09922=1218.466,-64.774,-38.748,179.770,5.388,149.009
C09923=1218.460,-64.524,-38.760,179.773,5.388,149.008
C09924=1218.456,-64.274,-38.772,179.775,5.389,149.007
C09925=1218.450,-64.025,-38.783,179.777,5.388,149.007
C09926=1218.446,-63.775,-38.795,179.780,5.389,149.006
C09927=1218.440,-63.525,-38.807,179.782,5.388,149.005
C09928=1218.435,-63.275,-38.818,179.785,5.389,149.005
C09929=1218.430,-63.026,-38.830,179.787,5.388,149.004
C09930=1218.424,-62.777,-38.842,179.789,5.389,149.003
C09931=1218.419,-62.527,-38.854,179.792,5.389,149.002
C09932=1218.414,-62.277,-38.865,179.794,5.389,149.002
C09933=1218.409,-62.027,-38.877,179.797,5.390,149.001
C09934=1218.403,-61.777,-38.889,179.799,5.389,149.000
C09935=1218.399,-61.528,-38.901,179.802,5.390,149.000
C09936=1218.393,-61.278,-38.913,179.804,5.390,148.999
C09937=1218.388,-61.028,-38.925,179.806,5.390,148.998
C09938=1218.383,-60.779,-38.936,179.809,5.391,148.998
C09939=1218.378,-60.530,-38.949,179.811,5.390,148.997
C09940=1218.373,-60.280,-38.961,179.813,5.391,148.996
C09941=1218.368,-60.030,-38.972,179.815,5.390,148.996
C09942=1218.363,-59.780,-38.984,179.818,5.391,148.995
C09943=1218.358,-59.531,-38.996,179.821,5.391,148.994
C09944=1218.352,-59.281,-39.008,179.823,5.391,148.994
C09945=1218.347,-59.031,-39.019,179.826,5.391,148.993
C09946=1218.342,-58.781,-39.031,179.828,5.391,148.992
C09947=1218.337,-58.532,-39.044,179.830,5.392,148.991
C09948=1218.332,-58.282,-39.055,179.833,5.392,148.991
C09949=1218.327,-58.032,-39.067,179.835,5.392,148.990
C09950=1218.322,-57.783,-39.080,179.838,5.392,148.989
C09951=1218.316,-57.533,-39.092,179.840,5.392,148.989
C09952=1218.312,-57.283,-39.103,179.842,5.392,148.988
C09953=1218.306,-57.034,-39.115,179.845,5.392,148.987
C09954=1218.301,-56.784,-39.127,179.847,5.392,148.986
C09955=1218.296,-56.534,-39.139,179.850,5.393,148.986
C09956=1218.291,-56.285,-39.151,179.851,5.393,148.985
C09957=1218.286,-56.035,-39.163,179.854,5.393,148.985
C09958=1218.280,-55.785,-39.175,179.856,5.393,148.984
C09959=1218.275,-55.536,-39.188,179.859,5.393,148.983
C09960=1218.270,-55.286,-39.200,179.862,5.394,148.983
C09961=1218.265,-55.037,-39.211,179.864,5.394,148.982
C09962=1218.260,-54.787,-39.223,179.866,5.394,148.981
C09963=1218.255,-54.537,-39.235,179.868,5.394,148.980
C09964=1218.249,-54.288,-39.248,179.871,5.394,148.980
C09965=1218.244,-54.038,-39.260,179.874,5.395,148.979
C09966=1218.239,-53.788,-39.271,179.876,5.394,148.978
C09967=1218.234,-53.539,-39.284,179.878,5.395,148.978
C09968=1218.229,-53.289,-39.296,179.881,5.394,148.977
C09969=1218.224,-53.040,-39.308,179.883,5.395,148.976
C09970=1218.218,-52.790,-39.320,179.886,5.395,148.975
C09971=1218.213,-52.541,-39.333,179.888,5.395,148.975
C09972=1218.208,-52.291,-39.344,179.891,5.395,148.974
C09973=1218.204,-52.041,-39.357,179.893,5.395,148.973
C09974=1218.198,-51.791,-39.369,179.895,5.396,148.973
C09975=1218.193,-51.542,-39.381,179.898,5.396,148.972
C09976=1218.188,-51.292,-39.393,179.900,5.396,148.971
C09977=1218.183,-51.042,-39.406,179.902,5.397,148.971
C09978=1218.177,-50.792,-39.418,179.905,5.397,148.970
C09979=1218.172,-50.543,-39.430,179.907,5.397,148.969
C09980=1218.167,-50.293,-39.442,179.910,5.397,148.969
C09981=1218.162,-50.044,-39.454,179.912,5.397,148.968
C09982=1218.157,-49.794,-39.466,179.914,5.397,148.967
C09983=1218.152,-49.545,-39.479,179.917,5.398,148.967
C09984=1218.146,-49.295,-39.491,179.919,5.397,148.966
C09985=1218.141,-49.025,-39.504,179.922,5.398,148.965
C09986=1218.135,-48.755,-39.518,179.925,5.398,148.964
C09987=1218.130,-48.486,-39.531,179.927,5.398,148.964
C09988=1218.124,-48.215,-39.544,179.930,5.398,148.963
C09989=1218.119,-47.966,-39.557,179.932,5.399,148.962
C09990=1218.114,-47.716,-39.569,179.935,5.398,148.961
C09991=1218.109,-47.467,-39.581,179.937,5.399,148.961
C09992=1218.104,-47.216,-39.593,179.940,5.399,148.960
C09993=1218.099,-46.967,-39.606,179.942,5.399,148.959
C09994=1218.094,-46.717,-39.619,179.945,5.399,148.959
C09995=1218.088,-46.467,-39.631,179.947,5.400,148.958
C09996=1218.083,-46.218,-39.643,179.949,5.400,148.957
//INST
///DATE 2021/06/15 17:22
///ATTR SC,RW,RJ
////FRAME ROBOT
///GROUP1 RB1
NOP
MOVL C00000 V=800.0 PL=0
MOVL C00001 V=800.0 PL=0
MOVL C00002 V=800.0 PL=0
MOVL C00003 V=800.0 PL=0
MOVL C00004 V=800.0 PL=0
MOVL C00005 V=800.0 PL=0
MOVL C00006 V=800.0 PL=0
MOVL C00007 V=800.0 PL=0
MOVL C00008 V=800.0 PL=0
MOVL C00009 V=800.0 PL=0
MOVL C00010 V=800.0 PL=0
MOVL C00011 V=800.0 PL=0
MOVL C00012 V=800.0 PL=0
MOVL C00013 V=800.0 PL=0
MOVL C00014 V=800.0 PL=0
MOVL C00015 V=800.0 PL=0
MOVL C00016 V=800.0 PL=0
MOVL C00017 V=800.0 PL=0
MOVL C00018 V=800.0 PL=0
MOVL C00019 V=800.0 PL=0
MOVL C00020 V=800.0 PL=0
MOVL C00021 V=800.0 PL=0
MOVL C00022 V=800.0 PL=0
MOVL C00023 V=800.0 PL=0
MOVL C00024 V=800.0 PL=0
MOVL C00025 V=800.0 PL=0
MOVL C00026 V=800.0 PL=0
MOVL C00027 V=800.0 PL=0
MOVL C00028 V=800.0 PL=0
MOVL C00029 V=800.0 PL=0
MOVL C00030 V=800.0 PL=0
MOVL C00031 V=800.0 PL=0
MOVL C00032 V=800.0 PL=0
MOVL C00033 V=800.0 PL=0
MOVL C00034 V=800.0 PL=0
MOVL C00035 V=800.0 PL=0
MOVL C00036 V=800.0 PL=0
MOVL C00037 V=800.0 PL=0
MOVL C00038 V=800.0 PL=0
MOVL C00039 V=800.0 PL=0
MOVL C00040 V=800.0 PL=0
MOVL C00041 V=800.0 PL=0
MOVL C00042 V=800.0 PL=0
MOVL C00043 V=800.0 PL=0
MOVL C00044 V=800.0 PL=0
MOVL C00045 V=800.0 PL=0
MOVL C00046 V=800.0 PL=0
MOVL C00047 V=800.0 PL=0
MOVL C00048 V=800.0 PL=0
MOVL C00049 V=800.0 PL=0
MOVL C00050 V=800.0 PL=0
MOVL C00051 V=800.0 PL=0
MOVL C00052 V=800.0 PL=0
MOVL C00053 V=800.0 PL=0
MOVL C00054 V=800.0 PL=0
MOVL C00055 V=800.0 PL=0
MOVL C00056 V=800.0 PL=0
MOVL C00057 V=800.0 PL=0
MOVL C00058 V=800.0 PL=0
MOVL C00059 V=800.0 PL=0
MOVL C00060 V=800.0 PL=0
MOVL C00061 V=800.0 PL=0
MOVL C00062 V=800.0 PL=0
MOVL C00063 V=800.0 PL=0
MOVL C00064 V=800.0 PL=0
MOVL C00065 V=800.0 PL=0
MOVL C00066 V=800.0 PL=0
MOVL C00067 V=800.0 PL=0
MOVL C00068 V=800.0 PL=0
MOVL C00069 V=800.0 PL=0
MOVL C00070 V=800.0 PL=0
MOVL C00071 V=800.0 PL=0
MOVL C00072 V=800.0 PL=0
MOVL C00073 V=800.0 PL=0
MOVL C00074 V=800.0 PL=0
MOVL C00075 V=800.0 PL=0
MOVL C00076 V=800.0 PL=0
MOVL C00077 V=800.0 PL=0
MOVL C00078 V=800.0 PL=0
MOVL C00079 V=800.0 PL=0
MOVL C00080 V=800.0 PL=0
MOVL C00081 V=800.0 PL=0
MOVL C00082 V=800.0 PL=0
MOVL C00083 V=800.0 PL=0
MOVL C00084 V=800.0 PL=0
MOVL C00085 V=800.0 PL=0
MOVL C00086 V=800.0 PL=0
MOVL C00087 V=800.0 PL=0
MOVL C00088 V=800.0 PL=0
MOVL C00089 V=800.0 PL=0
MOVL C00090 V=800.0 PL=0
MOVL C00091 V=800.0 PL=0
MOVL C00092 V=800.0 PL=0
MOVL C00093 V=800.0 PL=0
MOVL C00094 V=800.0 PL=0
MOVL C00095 V=800.0 PL=0
MOVL C00096 V=800.0 PL=0
MOVL C00097 V=800.0 PL=0
MOVL C00098 V=800.0 PL=0
MOVL C00099 V=800.0 PL=0
MOVL C00100 V=800.0 PL=0
MOVL C00101 V=800.0 PL=0
MOVL C00102 V=800.0 PL=0
MOVL C00103 V=800.0 PL=0
MOVL C00104 V=800.0 PL=0
MOVL C00105 V=800.0 PL=0
MOVL C00106 V=800.0 PL=0
MOVL C00107 V=800.0 PL=0
MOVL C00108 V=800.0 PL=0
MOVL C00109 V=800.0 PL=0
MOVL C00110 V=800.0 PL=0
MOVL C00111 V=800.0 PL=0
MOVL C00112 V=800.0 PL=0
MOVL C00113 V=800.0 PL=0
MOVL C00114 V=800.0 PL=0
MOVL C00115 V=800.0 PL=0
MOVL C00116 V=800.0 PL=0
MOVL C00117 V=800.0 PL=0
MOVL C00118 V=800.0 PL=0
MOVL C00119 V=800.0 PL=0
MOVL C00120 V=800.0 PL=0
MOVL C00121 V=800.0 PL=0
MOVL C00122 V=800.0 PL=0
MOVL C00123 V=800.0 PL=0
MOVL C00124 V=800.0 PL=0
MOVL C00125 V=800.0 PL=0
MOVL C00126 V=800.0 PL=0
MOVL C00127 V=800.0 PL=0
MOVL C00128 V=800.0 PL=0
MOVL C00129 V=800.0 PL=0
MOVL C00130 V=800.0 PL=0
MOVL C00131 V=800.0 PL=0
MOVL C00132 V=800.0 PL=0
MOVL C00133 V=800.0 PL=0
MOVL C00134 V=800.0 PL=0
MOVL C00135 V=800.0 PL=0
MOVL C00136 V=800.0 PL=0
MOVL C00137 V=800.0 PL=0
MOVL C00138 V=800.0 PL=0
MOVL C00139 V=800.0 PL=0
MOVL C00140 V=800.0 PL=0
MOVL C00141 V=800.0 PL=0
MOVL C00142 V=800.0 PL=0
MOVL C00143 V=800.0 PL=0
MOVL C00144 V=800.0 PL=0
MOVL C00145 V=800.0 PL=0
MOVL C00146 V=800.0 PL=0
MOVL C00147 V=800.0 PL=0
MOVL C00148 V=800.0 PL=0
MOVL C00149 V=800.0 PL=0
MOVL C00150 V=800.0 PL=0
MOVL C00151 V=800.0 PL=0
MOVL C00152 V=800.0 PL=0
MOVL C00153 V=800.0 PL=0
MOVL C00154 V=800.0 PL=0
MOVL C00155 V=800.0 PL=0
MOVL C00156 V=800.0 PL=0
MOVL C00157 V=800.0 PL=0
MOVL C00158 V=800.0 PL=0
MOVL C00159 V=800.0 PL=0
MOVL C00160 V=800.0 PL=0
MOVL C00161 V=800.0 PL=0
MOVL C00162 V=800.0 PL=0
MOVL C00163 V=800.0 PL=0
MOVL C00164 V=800.0 PL=0
MOVL C00165 V=800.0 PL=0
MOVL C00166 V=800.0 PL=0
MOVL C00167 V=800.0 PL=0
MOVL C00168 V=800.0 PL=0
MOVL C00169 V=800.0 PL=0
MOVL C00170 V=800.0 PL=0
MOVL C00171 V=800.0 PL=0
MOVL C00172 V=800.0 PL=0
MOVL C00173 V=800.0 PL=0
MOVL C00174 V=800.0 PL=0
MOVL C00175 V=800.0 PL=0
MOVL C00176 V=800.0 PL=0
MOVL C00177 V=800.0 PL=0
MOVL C00178 V=800.0 PL=0
MOVL C00179 V=800.0 PL=0
MOVL C00180 V=800.0 PL=0
MOVL C00181 V=800.0 PL=0
MOVL C00182 V=800.0 PL=0
MOVL C00183 V=800.0 PL=0
MOVL C00184 V=800.0 PL=0
MOVL C00185 V=800.0 PL=0
MOVL C00186 V=800.0 PL=0
MOVL C00187 V=800.0 PL=0
MOVL C00188 V=800.0 PL=0
MOVL C00189 V=800.0 PL=0
MOVL C00190 V=800.0 PL=0
MOVL C00191 V=800.0 PL=0
MOVL C00192 V=800.0 PL=0
MOVL C00193 V=800.0 PL=0
MOVL C00194 V=800.0 PL=0
MOVL C00195 V=800.0 PL=0
MOVL C00196 V=800.0 PL=0
MOVL C00197 V=800.0 PL=0
MOVL C00198 V=800.0 PL=0
MOVL C00199 V=800.0 PL=0
MOVL C00200 V=800.0 PL=0
MOVL C00201 V=800.0 PL=0
MOVL C00202 V=800.0 PL=0
MOVL C00203 V=800.0 PL=0
MOVL C00204 V=800.0 PL=0
MOVL C00205 V=800.0 PL=0
MOVL C00206 V=800.0 PL=0
MOVL C00207 V=800.0 PL=0
MOVL C00208 V=800.0 PL=0
MOVL C00209 V=800.0 PL=0
MOVL C00210 V=800.0 PL=0
MOVL C00211 V=800.0 PL=0
MOVL C00212 V=800.0 PL=0
MOVL C00213 V=800.0 PL=0
MOVL C00214 V=800.0 PL=0
MOVL C00215 V=800.0 PL=0
MOVL C00216 V=800.0 PL=0
MOVL C00217 V=800.0 PL=0
MOVL C00218 V=800.0 PL=0
MOVL C00219 V=800.0 PL=0
MOVL C00220 V=800.0 PL=0
MOVL C00221 V=800.0 PL=0
MOVL C00222 V=800.0 PL=0
MOVL C00223 V=800.0 PL=0
MOVL C00224 V=800.0 PL=0
MOVL C00225 V=800.0 PL=0
MOVL C00226 V=800.0 PL=0
MOVL C00227 V=800.0 PL=0
MOVL C00228 V=800.0 PL=0
MOVL C00229 V=800.0 PL=0
MOVL C00230 V=800.0 PL=0
MOVL C00231 V=800.0 PL=0
MOVL C00232 V=800.0 PL=0
MOVL C00233 V=800.0 PL=0
MOVL C00234 V=800.0 PL=0
MOVL C00235 V=800.0 PL=0
MOVL C00236 V=800.0 PL=0
MOVL C00237 V=800.0 PL=0
MOVL C00238 V=800.0 PL=0
MOVL C00239 V=800.0 PL=0
MOVL C00240 V=800.0 PL=0
MOVL C00241 V=800.0 PL=0
MOVL C00242 V=800.0 PL=0
MOVL C00243 V=800.0 PL=0
MOVL C00244 V=800.0 PL=0
MOVL C00245 V=800.0 PL=0
MOVL C00246 V=800.0 PL=0
MOVL C00247 V=800.0 PL=0
MOVL C00248 V=800.0 PL=0
MOVL C00249 V=800.0 PL=0
MOVL C00250 V=800.0 PL=0
MOVL C00251 V=800.0 PL=0
MOVL C00252 V=800.0 PL=0
MOVL C00253 V=800.0 PL=0
MOVL C00254 V=800.0 PL=0
MOVL C00255 V=800.0 PL=0
MOVL C00256 V=800.0 PL=0
MOVL C00257 V=800.0 PL=0
MOVL C00258 V=800.0 PL=0
MOVL C00259 V=800.0 PL=0
MOVL C00260 V=800.0 PL=0
MOVL C00261 V=800.0 PL=0
MOVL C00262 V=800.0 PL=0
MOVL C00263 V=800.0 PL=0
MOVL C00264 V=800.0 PL=0
MOVL C00265 V=800.0 PL=0
MOVL C00266 V=800.0 PL=0
MOVL C00267 V=800.0 PL=0
MOVL C00268 V=800.0 PL=0
MOVL C00269 V=800.0 PL=0
MOVL C00270 V=800.0 PL=0
MOVL C00271 V=800.0 PL=0
MOVL C00272 V=800.0 PL=0
MOVL C00273 V=800.0 PL=0
MOVL C00274 V=800.0 PL=0
MOVL C00275 V=800.0 PL=0
MOVL C00276 V=800.0 PL=0
MOVL C00277 V=800.0 PL=0
MOVL C00278 V=800.0 PL=0
MOVL C00279 V=800.0 PL=0
MOVL C00280 V=800.0 PL=0
MOVL C00281 V=800.0 PL=0
MOVL C00282 V=800.0 PL=0
MOVL C00283 V=800.0 PL=0
MOVL C00284 V=800.0 PL=0
MOVL C00285 V=800.0 PL=0
MOVL C00286 V=800.0 PL=0
MOVL C00287 V=800.0 PL=0
MOVL C00288 V=800.0 PL=0
MOVL C00289 V=800.0 PL=0
MOVL C00290 V=800.0 PL=0
MOVL C00291 V=800.0 PL=0
MOVL C00292 V=800.0 PL=0
MOVL C00293 V=800.0 PL=0
MOVL C00294 V=800.0 PL=0
MOVL C00295 V=800.0 PL=0
MOVL C00296 V=800.0 PL=0
MOVL C00297 V=800.0 PL=0
MOVL C00298 V=800.0 PL=0
MOVL C00299 V=800.0 PL=0
MOVL C00300 V=800.0 PL=0
MOVL C00301 V=800.0 PL=0
MOVL C00302 V=800.0 PL=0
MOVL C00303 V=800.0 PL=0
MOVL C00304 V=800.0 PL=0
MOVL C00305 V=800.0 PL=0
MOVL C00306 V=800.0 PL=0
MOVL C00307 V=800.0 PL=0
MOVL C00308 V=800.0 PL=0
MOVL C00309 V=800.0 PL=0
MOVL C00310 V=800.0 PL=0
MOVL C00311 V=800.0 PL=0
MOVL C00312 V=800.0 PL=0
MOVL C00313 V=800.0 PL=0
MOVL C00314 V=800.0 PL=0
MOVL C00315 V=800.0 PL=0
MOVL C00316 V=800.0 PL=0
MOVL C00317 V=800.0 PL=0
MOVL C00318 V=800.0 PL=0
MOVL C00319 V=800.0 PL=0
MOVL C00320 V=800.0 PL=0
MOVL C00321 V=800.0 PL=0
MOVL C00322 V=800.0 PL=0
MOVL C00323 V=800.0 PL=0
MOVL C00324 V=800.0 PL=0
MOVL C00325 V=800.0 PL=0
MOVL C00326 V=800.0 PL=0
MOVL C00327 V=800.0 PL=0
MOVL C00328 V=800.0 PL=0
MOVL C00329 V=800.0 PL=0
MOVL C00330 V=800.0 PL=0
MOVL C00331 V=800.0 PL=0
MOVL C00332 V=800.0 PL=0
MOVL C00333 V=800.0 PL=0
MOVL C00334 V=800.0 PL=0
MOVL C00335 V=800.0 PL=0
MOVL C00336 V=800.0 PL=0
MOVL C00337 V=800.0 PL=0
MOVL C00338 V=800.0 PL=0
MOVL C00339 V=800.0 PL=0
MOVL C00340 V=800.0 PL=0
MOVL C00341 V=800.0 PL=0
MOVL C00342 V=800.0 PL=0
MOVL C00343 V=800.0 PL=0
MOVL C00344 V=800.0 PL=0
MOVL C00345 V=800.0 PL=0
MOVL C00346 V=800.0 PL=0
MOVL C00347 V=800.0 PL=0
MOVL C00348 V=800.0 PL=0
MOVL C00349 V=800.0 PL=0
MOVL C00350 V=800.0 PL=0
MOVL C00351 V=800.0 PL=0
MOVL C00352 V=800.0 PL=0
MOVL C00353 V=800.0 PL=0
MOVL C00354 V=800.0 PL=0
MOVL C00355 V=800.0 PL=0
MOVL C00356 V=800.0 PL=0
MOVL C00357 V=800.0 PL=0
MOVL C00358 V=800.0 PL=0
MOVL C00359 V=800.0 PL=0
MOVL C00360 V=800.0 PL=0
MOVL C00361 V=800.0 PL=0
MOVL C00362 V=800.0 PL=0
MOVL C00363 V=800.0 PL=0
MOVL C00364 V=800.0 PL=0
MOVL C00365 V=800.0 PL=0
MOVL C00366 V=800.0 PL=0
MOVL C00367 V=800.0 PL=0
MOVL C00368 V=800.0 PL=0
MOVL C00369 V=800.0 PL=0
MOVL C00370 V=800.0 PL=0
MOVL C00371 V=800.0 PL=0
MOVL C00372 V=800.0 PL=0
MOVL C00373 V=800.0 PL=0
MOVL C00374 V=800.0 PL=0
MOVL C00375 V=800.0 PL=0
MOVL C00376 V=800.0 PL=0
MOVL C00377 V=800.0 PL=0
MOVL C00378 V=800.0 PL=0
MOVL C00379 V=800.0 PL=0
MOVL C00380 V=800.0 PL=0
MOVL C00381 V=800.0 PL=0
MOVL C00382 V=800.0 PL=0
MOVL C00383 V=800.0 PL=0
MOVL C00384 V=800.0 PL=0
MOVL C00385 V=800.0 PL=0
MOVL C00386 V=800.0 PL=0
MOVL C00387 V=800.0 PL=0
MOVL C00388 V=800.0 PL=0
MOVL C00389 V=800.0 PL=0
MOVL C00390 V=800.0 PL=0
MOVL C00391 V=800.0 PL=0
MOVL C00392 V=800.0 PL=0
MOVL C00393 V=800.0 PL=0
MOVL C00394 V=800.0 PL=0
MOVL C00395 V=800.0 PL=0
MOVL C00396 V=800.0 PL=0
MOVL C00397 V=800.0 PL=0
MOVL C00398 V=800.0 PL=0
MOVL C00399 V=800.0 PL=0
MOVL C00400 V=800.0 PL=0
MOVL C00401 V=800.0 PL=0
MOVL C00402 V=800.0 PL=0
MOVL C00403 V=800.0 PL=0
MOVL C00404 V=800.0 PL=0
MOVL C00405 V=800.0 PL=0
MOVL C00406 V=800.0 PL=0
MOVL C00407 V=800.0 PL=0
MOVL C00408 V=800.0 PL=0
MOVL C00409 V=800.0 PL=0
MOVL C00410 V=800.0 PL=0
MOVL C00411 V=800.0 PL=0
MOVL C00412 V=800.0 PL=0
MOVL C00413 V=800.0 PL=0
MOVL C00414 V=800.0 PL=0
MOVL C00415 V=800.0 PL=0
MOVL C00416 V=800.0 PL=0
MOVL C00417 V=800.0 PL=0
MOVL C00418 V=800.0 PL=0
MOVL C00419 V=800.0 PL=0
MOVL C00420 V=800.0 PL=0
MOVL C00421 V=800.0 PL=0
MOVL C00422 V=800.0 PL=0
MOVL C00423 V=800.0 PL=0
MOVL C00424 V=800.0 PL=0
MOVL C00425 V=800.0 PL=0
MOVL C00426 V=800.0 PL=0
MOVL C00427 V=800.0 PL=0
MOVL C00428 V=800.0 PL=0
MOVL C00429 V=800.0 PL=0
MOVL C00430 V=800.0 PL=0
MOVL C00431 V=800.0 PL=0
MOVL C00432 V=800.0 PL=0
MOVL C00433 V=800.0 PL=0
MOVL C00434 V=800.0 PL=0
MOVL C00435 V=800.0 PL=0
MOVL C00436 V=800.0 PL=0
MOVL C00437 V=800.0 PL=0
MOVL C00438 V=800.0 PL=0
MOVL C00439 V=800.0 PL=0
MOVL C00440 V=800.0 PL=0
MOVL C00441 V=800.0 PL=0
MOVL C00442 V=800.0 PL=0
MOVL C00443 V=800.0 PL=0
MOVL C00444 V=800.0 PL=0
MOVL C00445 V=800.0 PL=0
MOVL C00446 V=800.0 PL=0
MOVL C00447 V=800.0 PL=0
MOVL C00448 V=800.0 PL=0
MOVL C00449 V=800.0 PL=0
MOVL C00450 V=800.0 PL=0
MOVL C00451 V=800.0 PL=0
MOVL C00452 V=800.0 PL=0
MOVL C00453 V=800.0 PL=0
MOVL C00454 V=800.0 PL=0
MOVL C00455 V=800.0 PL=0
MOVL C00456 V=800.0 PL=0
MOVL C00457 V=800.0 PL=0
MOVL C00458 V=800.0 PL=0
MOVL C00459 V=800.0 PL=0
MOVL C00460 V=800.0 PL=0
MOVL C00461 V=800.0 PL=0
MOVL C00462 V=800.0 PL=0
MOVL C00463 V=800.0 PL=0
MOVL C00464 V=800.0 PL=0
MOVL C00465 V=800.0 PL=0
MOVL C00466 V=800.0 PL=0
MOVL C00467 V=800.0 PL=0
MOVL C00468 V=800.0 PL=0
MOVL C00469 V=800.0 PL=0
MOVL C00470 V=800.0 PL=0
MOVL C00471 V=800.0 PL=0
MOVL C00472 V=800.0 PL=0
MOVL C00473 V=800.0 PL=0
MOVL C00474 V=800.0 PL=0
MOVL C00475 V=800.0 PL=0
MOVL C00476 V=800.0 PL=0
MOVL C00477 V=800.0 PL=0
MOVL C00478 V=800.0 PL=0
MOVL C00479 V=800.0 PL=0
MOVL C00480 V=800.0 PL=0
MOVL C00481 V=800.0 PL=0
MOVL C00482 V=800.0 PL=0
MOVL C00483 V=800.0 PL=0
MOVL C00484 V=800.0 PL=0
MOVL C00485 V=800.0 PL=0
MOVL C00486 V=800.0 PL=0
MOVL C00487 V=800.0 PL=0
MOVL C00488 V=800.0 PL=0
MOVL C00489 V=800.0 PL=0
MOVL C00490 V=800.0 PL=0
MOVL C00491 V=800.0 PL=0
MOVL C00492 V=800.0 PL=0
MOVL C00493 V=800.0 PL=0
MOVL C00494 V=800.0 PL=0
MOVL C00495 V=800.0 PL=0
MOVL C00496 V=800.0 PL=0
MOVL C00497 V=800.0 PL=0
MOVL C00498 V=800.0 PL=0
MOVL C00499 V=800.0 PL=0
MOVL C00500 V=800.0 PL=0
MOVL C00501 V=800.0 PL=0
MOVL C00502 V=800.0 PL=0
MOVL C00503 V=800.0 PL=0
MOVL C00504 V=800.0 PL=0
MOVL C00505 V=800.0 PL=0
MOVL C00506 V=800.0 PL=0
MOVL C00507 V=800.0 PL=0
MOVL C00508 V=800.0 PL=0
MOVL C00509 V=800.0 PL=0
MOVL C00510 V=800.0 PL=0
MOVL C00511 V=800.0 PL=0
MOVL C00512 V=800.0 PL=0
MOVL C00513 V=800.0 PL=0
MOVL C00514 V=800.0 PL=0
MOVL C00515 V=800.0 PL=0
MOVL C00516 V=800.0 PL=0
MOVL C00517 V=800.0 PL=0
MOVL C00518 V=800.0 PL=0
MOVL C00519 V=800.0 PL=0
MOVL C00520 V=800.0 PL=0
MOVL C00521 V=800.0 PL=0
MOVL C00522 V=800.0 PL=0
MOVL C00523 V=800.0 PL=0
MOVL C00524 V=800.0 PL=0
MOVL C00525 V=800.0 PL=0
MOVL C00526 V=800.0 PL=0
MOVL C00527 V=800.0 PL=0
MOVL C00528 V=800.0 PL=0
MOVL C00529 V=800.0 PL=0
MOVL C00530 V=800.0 PL=0
MOVL C00531 V=800.0 PL=0
MOVL C00532 V=800.0 PL=0
MOVL C00533 V=800.0 PL=0
MOVL C00534 V=800.0 PL=0
MOVL C00535 V=800.0 PL=0
MOVL C00536 V=800.0 PL=0
MOVL C00537 V=800.0 PL=0
MOVL C00538 V=800.0 PL=0
MOVL C00539 V=800.0 PL=0
MOVL C00540 V=800.0 PL=0
MOVL C00541 V=800.0 PL=0
MOVL C00542 V=800.0 PL=0
MOVL C00543 V=800.0 PL=0
MOVL C00544 V=800.0 PL=0
MOVL C00545 V=800.0 PL=0
MOVL C00546 V=800.0 PL=0
MOVL C00547 V=800.0 PL=0
MOVL C00548 V=800.0 PL=0
MOVL C00549 V=800.0 PL=0
MOVL C00550 V=800.0 PL=0
MOVL C00551 V=800.0 PL=0
MOVL C00552 V=800.0 PL=0
MOVL C00553 V=800.0 PL=0
MOVL C00554 V=800.0 PL=0
MOVL C00555 V=800.0 PL=0
MOVL C00556 V=800.0 PL=0
MOVL C00557 V=800.0 PL=0
MOVL C00558 V=800.0 PL=0
MOVL C00559 V=800.0 PL=0
MOVL C00560 V=800.0 PL=0
MOVL C00561 V=800.0 PL=0
MOVL C00562 V=800.0 PL=0
MOVL C00563 V=800.0 PL=0
MOVL C00564 V=800.0 PL=0
MOVL C00565 V=800.0 PL=0
MOVL C00566 V=800.0 PL=0
MOVL C00567 V=800.0 PL=0
MOVL C00568 V=800.0 PL=0
MOVL C00569 V=800.0 PL=0
MOVL C00570 V=800.0 PL=0
MOVL C00571 V=800.0 PL=0
MOVL C00572 V=800.0 PL=0
MOVL C00573 V=800.0 PL=0
MOVL C00574 V=800.0 PL=0
MOVL C00575 V=800.0 PL=0
MOVL C00576 V=800.0 PL=0
MOVL C00577 V=800.0 PL=0
MOVL C00578 V=800.0 PL=0
MOVL C00579 V=800.0 PL=0
MOVL C00580 V=800.0 PL=0
MOVL C00581 V=800.0 PL=0
MOVL C00582 V=800.0 PL=0
MOVL C00583 V=800.0 PL=0
MOVL C00584 V=800.0 PL=0
MOVL C00585 V=800.0 PL=0
MOVL C00586 V=800.0 PL=0
MOVL C00587 V=800.0 PL=0
MOVL C00588 V=800.0 PL=0
MOVL C00589 V=800.0 PL=0
MOVL C00590 V=800.0 PL=0
MOVL C00591 V=800.0 PL=0
MOVL C00592 V=800.0 PL=0
MOVL C00593 V=800.0 PL=0
MOVL C00594 V=800.0 PL=0
MOVL C00595 V=800.0 PL=0
MOVL C00596 V=800.0 PL=0
MOVL C00597 V=800.0 PL=0
MOVL C00598 V=800.0 PL=0
MOVL C00599 V=800.0 PL=0
MOVL C00600 V=800.0 PL=0
MOVL C00601 V=800.0 PL=0
MOVL C00602 V=800.0 PL=0
MOVL C00603 V=800.0 PL=0
MOVL C00604 V=800.0 PL=0
MOVL C00605 V=800.0 PL=0
MOVL C00606 V=800.0 PL=0
MOVL C00607 V=800.0 PL=0
MOVL C00608 V=800.0 PL=0
MOVL C00609 V=800.0 PL=0
MOVL C00610 V=800.0 PL=0
MOVL C00611 V=800.0 PL=0
MOVL C00612 V=800.0 PL=0
MOVL C00613 V=800.0 PL=0
MOVL C00614 V=800.0 PL=0
MOVL C00615 V=800.0 PL=0
MOVL C00616 V=800.0 PL=0
MOVL C00617 V=800.0 PL=0
MOVL C00618 V=800.0 PL=0
MOVL C00619 V=800.0 PL=0
MOVL C00620 V=800.0 PL=0
MOVL C00621 V=800.0 PL=0
MOVL C00622 V=800.0 PL=0
MOVL C00623 V=800.0 PL=0
MOVL C00624 V=800.0 PL=0
MOVL C00625 V=800.0 PL=0
MOVL C00626 V=800.0 PL=0
MOVL C00627 V=800.0 PL=0
MOVL C00628 V=800.0 PL=0
MOVL C00629 V=800.0 PL=0
MOVL C00630 V=800.0 PL=0
MOVL C00631 V=800.0 PL=0
MOVL C00632 V=800.0 PL=0
MOVL C00633 V=800.0 PL=0
MOVL C00634 V=800.0 PL=0
MOVL C00635 V=800.0 PL=0
MOVL C00636 V=800.0 PL=0
MOVL C00637 V=800.0 PL=0
MOVL C00638 V=800.0 PL=0
MOVL C00639 V=800.0 PL=0
MOVL C00640 V=800.0 PL=0
MOVL C00641 V=800.0 PL=0
MOVL C00642 V=800.0 PL=0
MOVL C00643 V=800.0 PL=0
MOVL C00644 V=800.0 PL=0
MOVL C00645 V=800.0 PL=0
MOVL C00646 V=800.0 PL=0
MOVL C00647 V=800.0 PL=0
MOVL C00648 V=800.0 PL=0
MOVL C00649 V=800.0 PL=0
MOVL C00650 V=800.0 PL=0
MOVL C00651 V=800.0 PL=0
MOVL C00652 V=800.0 PL=0
MOVL C00653 V=800.0 PL=0
MOVL C00654 V=800.0 PL=0
MOVL C00655 V=800.0 PL=0
MOVL C00656 V=800.0 PL=0
MOVL C00657 V=800.0 PL=0
MOVL C00658 V=800.0 PL=0
MOVL C00659 V=800.0 PL=0
MOVL C00660 V=800.0 PL=0
MOVL C00661 V=800.0 PL=0
MOVL C00662 V=800.0 PL=0
MOVL C00663 V=800.0 PL=0
MOVL C00664 V=800.0 PL=0
MOVL C00665 V=800.0 PL=0
MOVL C00666 V=800.0 PL=0
MOVL C00667 V=800.0 PL=0
MOVL C00668 V=800.0 PL=0
MOVL C00669 V=800.0 PL=0
MOVL C00670 V=800.0 PL=0
MOVL C00671 V=800.0 PL=0
MOVL C00672 V=800.0 PL=0
MOVL C00673 V=800.0 PL=0
MOVL C00674 V=800.0 PL=0
MOVL C00675 V=800.0 PL=0
MOVL C00676 V=800.0 PL=0
MOVL C00677 V=800.0 PL=0
MOVL C00678 V=800.0 PL=0
MOVL C00679 V=800.0 PL=0
MOVL C00680 V=800.0 PL=0
MOVL C00681 V=800.0 PL=0
MOVL C00682 V=800.0 PL=0
MOVL C00683 V=800.0 PL=0
MOVL C00684 V=800.0 PL=0
MOVL C00685 V=800.0 PL=0
MOVL C00686 V=800.0 PL=0
MOVL C00687 V=800.0 PL=0
MOVL C00688 V=800.0 PL=0
MOVL C00689 V=800.0 PL=0
MOVL C00690 V=800.0 PL=0
MOVL C00691 V=800.0 PL=0
MOVL C00692 V=800.0 PL=0
MOVL C00693 V=800.0 PL=0
MOVL C00694 V=800.0 PL=0
MOVL C00695 V=800.0 PL=0
MOVL C00696 V=800.0 PL=0
MOVL C00697 V=800.0 PL=0
MOVL C00698 V=800.0 PL=0
MOVL C00699 V=800.0 PL=0
MOVL C00700 V=800.0 PL=0
MOVL C00701 V=800.0 PL=0
MOVL C00702 V=800.0 PL=0
MOVL C00703 V=800.0 PL=0
MOVL C00704 V=800.0 PL=0
MOVL C00705 V=800.0 PL=0
MOVL C00706 V=800.0 PL=0
MOVL C00707 V=800.0 PL=0
MOVL C00708 V=800.0 PL=0
MOVL C00709 V=800.0 PL=0
MOVL C00710 V=800.0 PL=0
MOVL C00711 V=800.0 PL=0
MOVL C00712 V=800.0 PL=0
MOVL C00713 V=800.0 PL=0
MOVL C00714 V=800.0 PL=0
MOVL C00715 V=800.0 PL=0
MOVL C00716 V=800.0 PL=0
MOVL C00717 V=800.0 PL=0
MOVL C00718 V=800.0 PL=0
MOVL C00719 V=800.0 PL=0
MOVL C00720 V=800.0 PL=0
MOVL C00721 V=800.0 PL=0
MOVL C00722 V=800.0 PL=0
MOVL C00723 V=800.0 PL=0
MOVL C00724 V=800.0 PL=0
MOVL C00725 V=800.0 PL=0
MOVL C00726 V=800.0 PL=0
MOVL C00727 V=800.0 PL=0
MOVL C00728 V=800.0 PL=0
MOVL C00729 V=800.0 PL=0
MOVL C00730 V=800.0 PL=0
MOVL C00731 V=800.0 PL=0
MOVL C00732 V=800.0 PL=0
MOVL C00733 V=800.0 PL=0
MOVL C00734 V=800.0 PL=0
MOVL C00735 V=800.0 PL=0
MOVL C00736 V=800.0 PL=0
MOVL C00737 V=800.0 PL=0
MOVL C00738 V=800.0 PL=0
MOVL C00739 V=800.0 PL=0
MOVL C00740 V=800.0 PL=0
MOVL C00741 V=800.0 PL=0
MOVL C00742 V=800.0 PL=0
MOVL C00743 V=800.0 PL=0
MOVL C00744 V=800.0 PL=0
MOVL C00745 V=800.0 PL=0
MOVL C00746 V=800.0 PL=0
MOVL C00747 V=800.0 PL=0
MOVL C00748 V=800.0 PL=0
MOVL C00749 V=800.0 PL=0
MOVL C00750 V=800.0 PL=0
MOVL C00751 V=800.0 PL=0
MOVL C00752 V=800.0 PL=0
MOVL C00753 V=800.0 PL=0
MOVL C00754 V=800.0 PL=0
MOVL C00755 V=800.0 PL=0
MOVL C00756 V=800.0 PL=0
MOVL C00757 V=800.0 PL=0
MOVL C00758 V=800.0 PL=0
MOVL C00759 V=800.0 PL=0
MOVL C00760 V=800.0 PL=0
MOVL C00761 V=800.0 PL=0
MOVL C00762 V=800.0 PL=0
MOVL C00763 V=800.0 PL=0
MOVL C00764 V=800.0 PL=0
MOVL C00765 V=800.0 PL=0
MOVL C00766 V=800.0 PL=0
MOVL C00767 V=800.0 PL=0
MOVL C00768 V=800.0 PL=0
MOVL C00769 V=800.0 PL=0
MOVL C00770 V=800.0 PL=0
MOVL C00771 V=800.0 PL=0
MOVL C00772 V=800.0 PL=0
MOVL C00773 V=800.0 PL=0
MOVL C00774 V=800.0 PL=0
MOVL C00775 V=800.0 PL=0
MOVL C00776 V=800.0 PL=0
MOVL C00777 V=800.0 PL=0
MOVL C00778 V=800.0 PL=0
MOVL C00779 V=800.0 PL=0
MOVL C00780 V=800.0 PL=0
MOVL C00781 V=800.0 PL=0
MOVL C00782 V=800.0 PL=0
MOVL C00783 V=800.0 PL=0
MOVL C00784 V=800.0 PL=0
MOVL C00785 V=800.0 PL=0
MOVL C00786 V=800.0 PL=0
MOVL C00787 V=800.0 PL=0
MOVL C00788 V=800.0 PL=0
MOVL C00789 V=800.0 PL=0
MOVL C00790 V=800.0 PL=0
MOVL C00791 V=800.0 PL=0
MOVL C00792 V=800.0 PL=0
MOVL C00793 V=800.0 PL=0
MOVL C00794 V=800.0 PL=0
MOVL C00795 V=800.0 PL=0
MOVL C00796 V=800.0 PL=0
MOVL C00797 V=800.0 PL=0
MOVL C00798 V=800.0 PL=0
MOVL C00799 V=800.0 PL=0
MOVL C00800 V=800.0 PL=0
MOVL C00801 V=800.0 PL=0
MOVL C00802 V=800.0 PL=0
MOVL C00803 V=800.0 PL=0
MOVL C00804 V=800.0 PL=0
MOVL C00805 V=800.0 PL=0
MOVL C00806 V=800.0 PL=0
MOVL C00807 V=800.0 PL=0
MOVL C00808 V=800.0 PL=0
MOVL C00809 V=800.0 PL=0
MOVL C00810 V=800.0 PL=0
MOVL C00811 V=800.0 PL=0
MOVL C00812 V=800.0 PL=0
MOVL C00813 V=800.0 PL=0
MOVL C00814 V=800.0 PL=0
MOVL C00815 V=800.0 PL=0
MOVL C00816 V=800.0 PL=0
MOVL C00817 V=800.0 PL=0
MOVL C00818 V=800.0 PL=0
MOVL C00819 V=800.0 PL=0
MOVL C00820 V=800.0 PL=0
MOVL C00821 V=800.0 PL=0
MOVL C00822 V=800.0 PL=0
MOVL C00823 V=800.0 PL=0
MOVL C00824 V=800.0 PL=0
MOVL C00825 V=800.0 PL=0
MOVL C00826 V=800.0 PL=0
MOVL C00827 V=800.0 PL=0
MOVL C00828 V=800.0 PL=0
MOVL C00829 V=800.0 PL=0
MOVL C00830 V=800.0 PL=0
MOVL C00831 V=800.0 PL=0
MOVL C00832 V=800.0 PL=0
MOVL C00833 V=800.0 PL=0
MOVL C00834 V=800.0 PL=0
MOVL C00835 V=800.0 PL=0
MOVL C00836 V=800.0 PL=0
MOVL C00837 V=800.0 PL=0
MOVL C00838 V=800.0 PL=0
MOVL C00839 V=800.0 PL=0
MOVL C00840 V=800.0 PL=0
MOVL C00841 V=800.0 PL=0
MOVL C00842 V=800.0 PL=0
MOVL C00843 V=800.0 PL=0
MOVL C00844 V=800.0 PL=0
MOVL C00845 V=800.0 PL=0
MOVL C00846 V=800.0 PL=0
MOVL C00847 V=800.0 PL=0
MOVL C00848 V=800.0 PL=0
MOVL C00849 V=800.0 PL=0
MOVL C00850 V=800.0 PL=0
MOVL C00851 V=800.0 PL=0
MOVL C00852 V=800.0 PL=0
MOVL C00853 V=800.0 PL=0
MOVL C00854 V=800.0 PL=0
MOVL C00855 V=800.0 PL=0
MOVL C00856 V=800.0 PL=0
MOVL C00857 V=800.0 PL=0
MOVL C00858 V=800.0 PL=0
MOVL C00859 V=800.0 PL=0
MOVL C00860 V=800.0 PL=0
MOVL C00861 V=800.0 PL=0
MOVL C00862 V=800.0 PL=0
MOVL C00863 V=800.0 PL=0
MOVL C00864 V=800.0 PL=0
MOVL C00865 V=800.0 PL=0
MOVL C00866 V=800.0 PL=0
MOVL C00867 V=800.0 PL=0
MOVL C00868 V=800.0 PL=0
MOVL C00869 V=800.0 PL=0
MOVL C00870 V=800.0 PL=0
MOVL C00871 V=800.0 PL=0
MOVL C00872 V=800.0 PL=0
MOVL C00873 V=800.0 PL=0
MOVL C00874 V=800.0 PL=0
MOVL C00875 V=800.0 PL=0
MOVL C00876 V=800.0 PL=0
MOVL C00877 V=800.0 PL=0
MOVL C00878 V=800.0 PL=0
MOVL C00879 V=800.0 PL=0
MOVL C00880 V=800.0 PL=0
MOVL C00881 V=800.0 PL=0
MOVL C00882 V=800.0 PL=0
MOVL C00883 V=800.0 PL=0
MOVL C00884 V=800.0 PL=0
MOVL C00885 V=800.0 PL=0
MOVL C00886 V=800.0 PL=0
MOVL C00887 V=800.0 PL=0
MOVL C00888 V=800.0 PL=0
MOVL C00889 V=800.0 PL=0
MOVL C00890 V=800.0 PL=0
MOVL C00891 V=800.0 PL=0
MOVL C00892 V=800.0 PL=0
MOVL C00893 V=800.0 PL=0
MOVL C00894 V=800.0 PL=0
MOVL C00895 V=800.0 PL=0
MOVL C00896 V=800.0 PL=0
MOVL C00897 V=800.0 PL=0
MOVL C00898 V=800.0 PL=0
MOVL C00899 V=800.0 PL=0
MOVL C00900 V=800.0 PL=0
MOVL C00901 V=800.0 PL=0
MOVL C00902 V=800.0 PL=0
MOVL C00903 V=800.0 PL=0
MOVL C00904 V=800.0 PL=0
MOVL C00905 V=800.0 PL=0
MOVL C00906 V=800.0 PL=0
MOVL C00907 V=800.0 PL=0
MOVL C00908 V=800.0 PL=0
MOVL C00909 V=800.0 PL=0
MOVL C00910 V=800.0 PL=0
MOVL C00911 V=800.0 PL=0
MOVL C00912 V=800.0 PL=0
MOVL C00913 V=800.0 PL=0
MOVL C00914 V=800.0 PL=0
MOVL C00915 V=800.0 PL=0
MOVL C00916 V=800.0 PL=0
MOVL C00917 V=800.0 PL=0
MOVL C00918 V=800.0 PL=0
MOVL C00919 V=800.0 PL=0
MOVL C00920 V=800.0 PL=0
MOVL C00921 V=800.0 PL=0
MOVL C00922 V=800.0 PL=0
MOVL C00923 V=800.0 PL=0
MOVL C00924 V=800.0 PL=0
MOVL C00925 V=800.0 PL=0
MOVL C00926 V=800.0 PL=0
MOVL C00927 V=800.0 PL=0
MOVL C00928 V=800.0 PL=0
MOVL C00929 V=800.0 PL=0
MOVL C00930 V=800.0 PL=0
MOVL C00931 V=800.0 PL=0
MOVL C00932 V=800.0 PL=0
MOVL C00933 V=800.0 PL=0
MOVL C00934 V=800.0 PL=0
MOVL C00935 V=800.0 PL=0
MOVL C00936 V=800.0 PL=0
MOVL C00937 V=800.0 PL=0
MOVL C00938 V=800.0 PL=0
MOVL C00939 V=800.0 PL=0
MOVL C00940 V=800.0 PL=0
MOVL C00941 V=800.0 PL=0
MOVL C00942 V=800.0 PL=0
MOVL C00943 V=800.0 PL=0
MOVL C00944 V=800.0 PL=0
MOVL C00945 V=800.0 PL=0
MOVL C00946 V=800.0 PL=0
MOVL C00947 V=800.0 PL=0
MOVL C00948 V=800.0 PL=0
MOVL C00949 V=800.0 PL=0
MOVL C00950 V=800.0 PL=0
MOVL C00951 V=800.0 PL=0
MOVL C00952 V=800.0 PL=0
MOVL C00953 V=800.0 PL=0
MOVL C00954 V=800.0 PL=0
MOVL C00955 V=800.0 PL=0
MOVL C00956 V=800.0 PL=0
MOVL C00957 V=800.0 PL=0
MOVL C00958 V=800.0 PL=0
MOVL C00959 V=800.0 PL=0
MOVL C00960 V=800.0 PL=0
MOVL C00961 V=800.0 PL=0
MOVL C00962 V=800.0 PL=0
MOVL C00963 V=800.0 PL=0
MOVL C00964 V=800.0 PL=0
MOVL C00965 V=800.0 PL=0
MOVL C00966 V=800.0 PL=0
MOVL C00967 V=800.0 PL=0
MOVL C00968 V=800.0 PL=0
MOVL C00969 V=800.0 PL=0
MOVL C00970 V=800.0 PL=0
MOVL C00971 V=800.0 PL=0
MOVL C00972 V=800.0 PL=0
MOVL C00973 V=800.0 PL=0
MOVL C00974 V=800.0 PL=0
MOVL C00975 V=800.0 PL=0
MOVL C00976 V=800.0 PL=0
MOVL C00977 V=800.0 PL=0
MOVL C00978 V=800.0 PL=0
MOVL C00979 V=800.0 PL=0
MOVL C00980 V=800.0 PL=0
MOVL C00981 V=800.0 PL=0
MOVL C00982 V=800.0 PL=0
MOVL C00983 V=800.0 PL=0
MOVL C00984 V=800.0 PL=0
MOVL C00985 V=800.0 PL=0
MOVL C00986 V=800.0 PL=0
MOVL C00987 V=800.0 PL=0
MOVL C00988 V=800.0 PL=0
MOVL C00989 V=800.0 PL=0
MOVL C00990 V=800.0 PL=0
MOVL C00991 V=800.0 PL=0
MOVL C00992 V=800.0 PL=0
MOVL C00993 V=800.0 PL=0
MOVL C00994 V=800.0 PL=0
MOVL C00995 V=800.0 PL=0
MOVL C00996 V=800.0 PL=0
MOVL C00997 V=800.0 PL=0
MOVL C00998 V=800.0 PL=0
MOVL C00999 V=800.0 PL=0
MOVL C01000 V=800.0 PL=0
MOVL C01001 V=800.0 PL=0
MOVL C01002 V=800.0 PL=0
MOVL C01003 V=800.0 PL=0
MOVL C01004 V=800.0 PL=0
MOVL C01005 V=800.0 PL=0
MOVL C01006 V=800.0 PL=0
MOVL C01007 V=800.0 PL=0
MOVL C01008 V=800.0 PL=0
MOVL C01009 V=800.0 PL=0
MOVL C01010 V=800.0 PL=0
MOVL C01011 V=800.0 PL=0
MOVL C01012 V=800.0 PL=0
MOVL C01013 V=800.0 PL=0
MOVL C01014 V=800.0 PL=0
MOVL C01015 V=800.0 PL=0
MOVL C01016 V=800.0 PL=0
MOVL C01017 V=800.0 PL=0
MOVL C01018 V=800.0 PL=0
MOVL C01019 V=800.0 PL=0
MOVL C01020 V=800.0 PL=0
MOVL C01021 V=800.0 PL=0
MOVL C01022 V=800.0 PL=0
MOVL C01023 V=800.0 PL=0
MOVL C01024 V=800.0 PL=0
MOVL C01025 V=800.0 PL=0
MOVL C01026 V=800.0 PL=0
MOVL C01027 V=800.0 PL=0
MOVL C01028 V=800.0 PL=0
MOVL C01029 V=800.0 PL=0
MOVL C01030 V=800.0 PL=0
MOVL C01031 V=800.0 PL=0
MOVL C01032 V=800.0 PL=0
MOVL C01033 V=800.0 PL=0
MOVL C01034 V=800.0 PL=0
MOVL C01035 V=800.0 PL=0
MOVL C01036 V=800.0 PL=0
MOVL C01037 V=800.0 PL=0
MOVL C01038 V=800.0 PL=0
MOVL C01039 V=800.0 PL=0
MOVL C01040 V=800.0 PL=0
MOVL C01041 V=800.0 PL=0
MOVL C01042 V=800.0 PL=0
MOVL C01043 V=800.0 PL=0
MOVL C01044 V=800.0 PL=0
MOVL C01045 V=800.0 PL=0
MOVL C01046 V=800.0 PL=0
MOVL C01047 V=800.0 PL=0
MOVL C01048 V=800.0 PL=0
MOVL C01049 V=800.0 PL=0
MOVL C01050 V=800.0 PL=0
MOVL C01051 V=800.0 PL=0
MOVL C01052 V=800.0 PL=0
MOVL C01053 V=800.0 PL=0
MOVL C01054 V=800.0 PL=0
MOVL C01055 V=800.0 PL=0
MOVL C01056 V=800.0 PL=0
MOVL C01057 V=800.0 PL=0
MOVL C01058 V=800.0 PL=0
MOVL C01059 V=800.0 PL=0
MOVL C01060 V=800.0 PL=0
MOVL C01061 V=800.0 PL=0
MOVL C01062 V=800.0 PL=0
MOVL C01063 V=800.0 PL=0
MOVL C01064 V=800.0 PL=0
MOVL C01065 V=800.0 PL=0
MOVL C01066 V=800.0 PL=0
MOVL C01067 V=800.0 PL=0
MOVL C01068 V=800.0 PL=0
MOVL C01069 V=800.0 PL=0
MOVL C01070 V=800.0 PL=0
MOVL C01071 V=800.0 PL=0
MOVL C01072 V=800.0 PL=0
MOVL C01073 V=800.0 PL=0
MOVL C01074 V=800.0 PL=0
MOVL C01075 V=800.0 PL=0
MOVL C01076 V=800.0 PL=0
MOVL C01077 V=800.0 PL=0
MOVL C01078 V=800.0 PL=0
MOVL C01079 V=800.0 PL=0
MOVL C01080 V=800.0 PL=0
MOVL C01081 V=800.0 PL=0
MOVL C01082 V=800.0 PL=0
MOVL C01083 V=800.0 PL=0
MOVL C01084 V=800.0 PL=0
MOVL C01085 V=800.0 PL=0
MOVL C01086 V=800.0 PL=0
MOVL C01087 V=800.0 PL=0
MOVL C01088 V=800.0 PL=0
MOVL C01089 V=800.0 PL=0
MOVL C01090 V=800.0 PL=0
MOVL C01091 V=800.0 PL=0
MOVL C01092 V=800.0 PL=0
MOVL C01093 V=800.0 PL=0
MOVL C01094 V=800.0 PL=0
MOVL C01095 V=800.0 PL=0
MOVL C01096 V=800.0 PL=0
MOVL C01097 V=800.0 PL=0
MOVL C01098 V=800.0 PL=0
MOVL C01099 V=800.0 PL=0
MOVL C01100 V=800.0 PL=0
MOVL C01101 V=800.0 PL=0
MOVL C01102 V=800.0 PL=0
MOVL C01103 V=800.0 PL=0
MOVL C01104 V=800.0 PL=0
MOVL C01105 V=800.0 PL=0
MOVL C01106 V=800.0 PL=0
MOVL C01107 V=800.0 PL=0
MOVL C01108 V=800.0 PL=0
MOVL C01109 V=800.0 PL=0
MOVL C01110 V=800.0 PL=0
MOVL C01111 V=800.0 PL=0
MOVL C01112 V=800.0 PL=0
MOVL C01113 V=800.0 PL=0
MOVL C01114 V=800.0 PL=0
MOVL C01115 V=800.0 PL=0
MOVL C01116 V=800.0 PL=0
MOVL C01117 V=800.0 PL=0
MOVL C01118 V=800.0 PL=0
MOVL C01119 V=800.0 PL=0
MOVL C01120 V=800.0 PL=0
MOVL C01121 V=800.0 PL=0
MOVL C01122 V=800.0 PL=0
MOVL C01123 V=800.0 PL=0
MOVL C01124 V=800.0 PL=0
MOVL C01125 V=800.0 PL=0
MOVL C01126 V=800.0 PL=0
MOVL C01127 V=800.0 PL=0
MOVL C01128 V=800.0 PL=0
MOVL C01129 V=800.0 PL=0
MOVL C01130 V=800.0 PL=0
MOVL C01131 V=800.0 PL=0
MOVL C01132 V=800.0 PL=0
MOVL C01133 V=800.0 PL=0
MOVL C01134 V=800.0 PL=0
MOVL C01135 V=800.0 PL=0
MOVL C01136 V=800.0 PL=0
MOVL C01137 V=800.0 PL=0
MOVL C01138 V=800.0 PL=0
MOVL C01139 V=800.0 PL=0
MOVL C01140 V=800.0 PL=0
MOVL C01141 V=800.0 PL=0
MOVL C01142 V=800.0 PL=0
MOVL C01143 V=800.0 PL=0
MOVL C01144 V=800.0 PL=0
MOVL C01145 V=800.0 PL=0
MOVL C01146 V=800.0 PL=0
MOVL C01147 V=800.0 PL=0
MOVL C01148 V=800.0 PL=0
MOVL C01149 V=800.0 PL=0
MOVL C01150 V=800.0 PL=0
MOVL C01151 V=800.0 PL=0
MOVL C01152 V=800.0 PL=0
MOVL C01153 V=800.0 PL=0
MOVL C01154 V=800.0 PL=0
MOVL C01155 V=800.0 PL=0
MOVL C01156 V=800.0 PL=0
MOVL C01157 V=800.0 PL=0
MOVL C01158 V=800.0 PL=0
MOVL C01159 V=800.0 PL=0
MOVL C01160 V=800.0 PL=0
MOVL C01161 V=800.0 PL=0
MOVL C01162 V=800.0 PL=0
MOVL C01163 V=800.0 PL=0
MOVL C01164 V=800.0 PL=0
MOVL C01165 V=800.0 PL=0
MOVL C01166 V=800.0 PL=0
MOVL C01167 V=800.0 PL=0
MOVL C01168 V=800.0 PL=0
MOVL C01169 V=800.0 PL=0
MOVL C01170 V=800.0 PL=0
MOVL C01171 V=800.0 PL=0
MOVL C01172 V=800.0 PL=0
MOVL C01173 V=800.0 PL=0
MOVL C01174 V=800.0 PL=0
MOVL C01175 V=800.0 PL=0
MOVL C01176 V=800.0 PL=0
MOVL C01177 V=800.0 PL=0
MOVL C01178 V=800.0 PL=0
MOVL C01179 V=800.0 PL=0
MOVL C01180 V=800.0 PL=0
MOVL C01181 V=800.0 PL=0
MOVL C01182 V=800.0 PL=0
MOVL C01183 V=800.0 PL=0
MOVL C01184 V=800.0 PL=0
MOVL C01185 V=800.0 PL=0
MOVL C01186 V=800.0 PL=0
MOVL C01187 V=800.0 PL=0
MOVL C01188 V=800.0 PL=0
MOVL C01189 V=800.0 PL=0
MOVL C01190 V=800.0 PL=0
MOVL C01191 V=800.0 PL=0
MOVL C01192 V=800.0 PL=0
MOVL C01193 V=800.0 PL=0
MOVL C01194 V=800.0 PL=0
MOVL C01195 V=800.0 PL=0
MOVL C01196 V=800.0 PL=0
MOVL C01197 V=800.0 PL=0
MOVL C01198 V=800.0 PL=0
MOVL C01199 V=800.0 PL=0
MOVL C01200 V=800.0 PL=0
MOVL C01201 V=800.0 PL=0
MOVL C01202 V=800.0 PL=0
MOVL C01203 V=800.0 PL=0
MOVL C01204 V=800.0 PL=0
MOVL C01205 V=800.0 PL=0
MOVL C01206 V=800.0 PL=0
MOVL C01207 V=800.0 PL=0
MOVL C01208 V=800.0 PL=0
MOVL C01209 V=800.0 PL=0
MOVL C01210 V=800.0 PL=0
MOVL C01211 V=800.0 PL=0
MOVL C01212 V=800.0 PL=0
MOVL C01213 V=800.0 PL=0
MOVL C01214 V=800.0 PL=0
MOVL C01215 V=800.0 PL=0
MOVL C01216 V=800.0 PL=0
MOVL C01217 V=800.0 PL=0
MOVL C01218 V=800.0 PL=0
MOVL C01219 V=800.0 PL=0
MOVL C01220 V=800.0 PL=0
MOVL C01221 V=800.0 PL=0
MOVL C01222 V=800.0 PL=0
MOVL C01223 V=800.0 PL=0
MOVL C01224 V=800.0 PL=0
MOVL C01225 V=800.0 PL=0
MOVL C01226 V=800.0 PL=0
MOVL C01227 V=800.0 PL=0
MOVL C01228 V=800.0 PL=0
MOVL C01229 V=800.0 PL=0
MOVL C01230 V=800.0 PL=0
MOVL C01231 V=800.0 PL=0
MOVL C01232 V=800.0 PL=0
MOVL C01233 V=800.0 PL=0
MOVL C01234 V=800.0 PL=0
MOVL C01235 V=800.0 PL=0
MOVL C01236 V=800.0 PL=0
MOVL C01237 V=800.0 PL=0
MOVL C01238 V=800.0 PL=0
MOVL C01239 V=800.0 PL=0
MOVL C01240 V=800.0 PL=0
MOVL C01241 V=800.0 PL=0
MOVL C01242 V=800.0 PL=0
MOVL C01243 V=800.0 PL=0
MOVL C01244 V=800.0 PL=0
MOVL C01245 V=800.0 PL=0
MOVL C01246 V=800.0 PL=0
MOVL C01247 V=800.0 PL=0
MOVL C01248 V=800.0 PL=0
MOVL C01249 V=800.0 PL=0
MOVL C01250 V=800.0 PL=0
MOVL C01251 V=800.0 PL=0
MOVL C01252 V=800.0 PL=0
MOVL C01253 V=800.0 PL=0
MOVL C01254 V=800.0 PL=0
MOVL C01255 V=800.0 PL=0
MOVL C01256 V=800.0 PL=0
MOVL C01257 V=800.0 PL=0
MOVL C01258 V=800.0 PL=0
MOVL C01259 V=800.0 PL=0
MOVL C01260 V=800.0 PL=0
MOVL C01261 V=800.0 PL=0
MOVL C01262 V=800.0 PL=0
MOVL C01263 V=800.0 PL=0
MOVL C01264 V=800.0 PL=0
MOVL C01265 V=800.0 PL=0
MOVL C01266 V=800.0 PL=0
MOVL C01267 V=800.0 PL=0
MOVL C01268 V=800.0 PL=0
MOVL C01269 V=800.0 PL=0
MOVL C01270 V=800.0 PL=0
MOVL C01271 V=800.0 PL=0
MOVL C01272 V=800.0 PL=0
MOVL C01273 V=800.0 PL=0
MOVL C01274 V=800.0 PL=0
MOVL C01275 V=800.0 PL=0
MOVL C01276 V=800.0 PL=0
MOVL C01277 V=800.0 PL=0
MOVL C01278 V=800.0 PL=0
MOVL C01279 V=800.0 PL=0
MOVL C01280 V=800.0 PL=0
MOVL C01281 V=800.0 PL=0
MOVL C01282 V=800.0 PL=0
MOVL C01283 V=800.0 PL=0
MOVL C01284 V=800.0 PL=0
MOVL C01285 V=800.0 PL=0
MOVL C01286 V=800.0 PL=0
MOVL C01287 V=800.0 PL=0
MOVL C01288 V=800.0 PL=0
MOVL C01289 V=800.0 PL=0
MOVL C01290 V=800.0 PL=0
MOVL C01291 V=800.0 PL=0
MOVL C01292 V=800.0 PL=0
MOVL C01293 V=800.0 PL=0
MOVL C01294 V=800.0 PL=0
MOVL C01295 V=800.0 PL=0
MOVL C01296 V=800.0 PL=0
MOVL C01297 V=800.0 PL=0
MOVL C01298 V=800.0 PL=0
MOVL C01299 V=800.0 PL=0
MOVL C01300 V=800.0 PL=0
MOVL C01301 V=800.0 PL=0
MOVL C01302 V=800.0 PL=0
MOVL C01303 V=800.0 PL=0
MOVL C01304 V=800.0 PL=0
MOVL C01305 V=800.0 PL=0
MOVL C01306 V=800.0 PL=0
MOVL C01307 V=800.0 PL=0
MOVL C01308 V=800.0 PL=0
MOVL C01309 V=800.0 PL=0
MOVL C01310 V=800.0 PL=0
MOVL C01311 V=800.0 PL=0
MOVL C01312 V=800.0 PL=0
MOVL C01313 V=800.0 PL=0
MOVL C01314 V=800.0 PL=0
MOVL C01315 V=800.0 PL=0
MOVL C01316 V=800.0 PL=0
MOVL C01317 V=800.0 PL=0
MOVL C01318 V=800.0 PL=0
MOVL C01319 V=800.0 PL=0
MOVL C01320 V=800.0 PL=0
MOVL C01321 V=800.0 PL=0
MOVL C01322 V=800.0 PL=0
MOVL C01323 V=800.0 PL=0
MOVL C01324 V=800.0 PL=0
MOVL C01325 V=800.0 PL=0
MOVL C01326 V=800.0 PL=0
MOVL C01327 V=800.0 PL=0
MOVL C01328 V=800.0 PL=0
MOVL C01329 V=800.0 PL=0
MOVL C01330 V=800.0 PL=0
MOVL C01331 V=800.0 PL=0
MOVL C01332 V=800.0 PL=0
MOVL C01333 V=800.0 PL=0
MOVL C01334 V=800.0 PL=0
MOVL C01335 V=800.0 PL=0
MOVL C01336 V=800.0 PL=0
MOVL C01337 V=800.0 PL=0
MOVL C01338 V=800.0 PL=0
MOVL C01339 V=800.0 PL=0
MOVL C01340 V=800.0 PL=0
MOVL C01341 V=800.0 PL=0
MOVL C01342 V=800.0 PL=0
MOVL C01343 V=800.0 PL=0
MOVL C01344 V=800.0 PL=0
MOVL C01345 V=800.0 PL=0
MOVL C01346 V=800.0 PL=0
MOVL C01347 V=800.0 PL=0
MOVL C01348 V=800.0 PL=0
MOVL C01349 V=800.0 PL=0
MOVL C01350 V=800.0 PL=0
MOVL C01351 V=800.0 PL=0
MOVL C01352 V=800.0 PL=0
MOVL C01353 V=800.0 PL=0
MOVL C01354 V=800.0 PL=0
MOVL C01355 V=800.0 PL=0
MOVL C01356 V=800.0 PL=0
MOVL C01357 V=800.0 PL=0
MOVL C01358 V=800.0 PL=0
MOVL C01359 V=800.0 PL=0
MOVL C01360 V=800.0 PL=0
MOVL C01361 V=800.0 PL=0
MOVL C01362 V=800.0 PL=0
MOVL C01363 V=800.0 PL=0
MOVL C01364 V=800.0 PL=0
MOVL C01365 V=800.0 PL=0
MOVL C01366 V=800.0 PL=0
MOVL C01367 V=800.0 PL=0
MOVL C01368 V=800.0 PL=0
MOVL C01369 V=800.0 PL=0
MOVL C01370 V=800.0 PL=0
MOVL C01371 V=800.0 PL=0
MOVL C01372 V=800.0 PL=0
MOVL C01373 V=800.0 PL=0
MOVL C01374 V=800.0 PL=0
MOVL C01375 V=800.0 PL=0
MOVL C01376 V=800.0 PL=0
MOVL C01377 V=800.0 PL=0
MOVL C01378 V=800.0 PL=0
MOVL C01379 V=800.0 PL=0
MOVL C01380 V=800.0 PL=0
MOVL C01381 V=800.0 PL=0
MOVL C01382 V=800.0 PL=0
MOVL C01383 V=800.0 PL=0
MOVL C01384 V=800.0 PL=0
MOVL C01385 V=800.0 PL=0
MOVL C01386 V=800.0 PL=0
MOVL C01387 V=800.0 PL=0
MOVL C01388 V=800.0 PL=0
MOVL C01389 V=800.0 PL=0
MOVL C01390 V=800.0 PL=0
MOVL C01391 V=800.0 PL=0
MOVL C01392 V=800.0 PL=0
MOVL C01393 V=800.0 PL=0
MOVL C01394 V=800.0 PL=0
MOVL C01395 V=800.0 PL=0
MOVL C01396 V=800.0 PL=0
MOVL C01397 V=800.0 PL=0
MOVL C01398 V=800.0 PL=0
MOVL C01399 V=800.0 PL=0
MOVL C01400 V=800.0 PL=0
MOVL C01401 V=800.0 PL=0
MOVL C01402 V=800.0 PL=0
MOVL C01403 V=800.0 PL=0
MOVL C01404 V=800.0 PL=0
MOVL C01405 V=800.0 PL=0
MOVL C01406 V=800.0 PL=0
MOVL C01407 V=800.0 PL=0
MOVL C01408 V=800.0 PL=0
MOVL C01409 V=800.0 PL=0
MOVL C01410 V=800.0 PL=0
MOVL C01411 V=800.0 PL=0
MOVL C01412 V=800.0 PL=0
MOVL C01413 V=800.0 PL=0
MOVL C01414 V=800.0 PL=0
MOVL C01415 V=800.0 PL=0
MOVL C01416 V=800.0 PL=0
MOVL C01417 V=800.0 PL=0
MOVL C01418 V=800.0 PL=0
MOVL C01419 V=800.0 PL=0
MOVL C01420 V=800.0 PL=0
MOVL C01421 V=800.0 PL=0
MOVL C01422 V=800.0 PL=0
MOVL C01423 V=800.0 PL=0
MOVL C01424 V=800.0 PL=0
MOVL C01425 V=800.0 PL=0
MOVL C01426 V=800.0 PL=0
MOVL C01427 V=800.0 PL=0
MOVL C01428 V=800.0 PL=0
MOVL C01429 V=800.0 PL=0
MOVL C01430 V=800.0 PL=0
MOVL C01431 V=800.0 PL=0
MOVL C01432 V=800.0 PL=0
MOVL C01433 V=800.0 PL=0
MOVL C01434 V=800.0 PL=0
MOVL C01435 V=800.0 PL=0
MOVL C01436 V=800.0 PL=0
MOVL C01437 V=800.0 PL=0
MOVL C01438 V=800.0 PL=0
MOVL C01439 V=800.0 PL=0
MOVL C01440 V=800.0 PL=0
MOVL C01441 V=800.0 PL=0
MOVL C01442 V=800.0 PL=0
MOVL C01443 V=800.0 PL=0
MOVL C01444 V=800.0 PL=0
MOVL C01445 V=800.0 PL=0
MOVL C01446 V=800.0 PL=0
MOVL C01447 V=800.0 PL=0
MOVL C01448 V=800.0 PL=0
MOVL C01449 V=800.0 PL=0
MOVL C01450 V=800.0 PL=0
MOVL C01451 V=800.0 PL=0
MOVL C01452 V=800.0 PL=0
MOVL C01453 V=800.0 PL=0
MOVL C01454 V=800.0 PL=0
MOVL C01455 V=800.0 PL=0
MOVL C01456 V=800.0 PL=0
MOVL C01457 V=800.0 PL=0
MOVL C01458 V=800.0 PL=0
MOVL C01459 V=800.0 PL=0
MOVL C01460 V=800.0 PL=0
MOVL C01461 V=800.0 PL=0
MOVL C01462 V=800.0 PL=0
MOVL C01463 V=800.0 PL=0
MOVL C01464 V=800.0 PL=0
MOVL C01465 V=800.0 PL=0
MOVL C01466 V=800.0 PL=0
MOVL C01467 V=800.0 PL=0
MOVL C01468 V=800.0 PL=0
MOVL C01469 V=800.0 PL=0
MOVL C01470 V=800.0 PL=0
MOVL C01471 V=800.0 PL=0
MOVL C01472 V=800.0 PL=0
MOVL C01473 V=800.0 PL=0
MOVL C01474 V=800.0 PL=0
MOVL C01475 V=800.0 PL=0
MOVL C01476 V=800.0 PL=0
MOVL C01477 V=800.0 PL=0
MOVL C01478 V=800.0 PL=0
MOVL C01479 V=800.0 PL=0
MOVL C01480 V=800.0 PL=0
MOVL C01481 V=800.0 PL=0
MOVL C01482 V=800.0 PL=0
MOVL C01483 V=800.0 PL=0
MOVL C01484 V=800.0 PL=0
MOVL C01485 V=800.0 PL=0
MOVL C01486 V=800.0 PL=0
MOVL C01487 V=800.0 PL=0
MOVL C01488 V=800.0 PL=0
MOVL C01489 V=800.0 PL=0
MOVL C01490 V=800.0 PL=0
MOVL C01491 V=800.0 PL=0
MOVL C01492 V=800.0 PL=0
MOVL C01493 V=800.0 PL=0
MOVL C01494 V=800.0 PL=0
MOVL C01495 V=800.0 PL=0
MOVL C01496 V=800.0 PL=0
MOVL C01497 V=800.0 PL=0
MOVL C01498 V=800.0 PL=0
MOVL C01499 V=800.0 PL=0
MOVL C01500 V=800.0 PL=0
MOVL C01501 V=800.0 PL=0
MOVL C01502 V=800.0 PL=0
MOVL C01503 V=800.0 PL=0
MOVL C01504 V=800.0 PL=0
MOVL C01505 V=800.0 PL=0
MOVL C01506 V=800.0 PL=0
MOVL C01507 V=800.0 PL=0
MOVL C01508 V=800.0 PL=0
MOVL C01509 V=800.0 PL=0
MOVL C01510 V=800.0 PL=0
MOVL C01511 V=800.0 PL=0
MOVL C01512 V=800.0 PL=0
MOVL C01513 V=800.0 PL=0
MOVL C01514 V=800.0 PL=0
MOVL C01515 V=800.0 PL=0
MOVL C01516 V=800.0 PL=0
MOVL C01517 V=800.0 PL=0
MOVL C01518 V=800.0 PL=0
MOVL C01519 V=800.0 PL=0
MOVL C01520 V=800.0 PL=0
MOVL C01521 V=800.0 PL=0
MOVL C01522 V=800.0 PL=0
MOVL C01523 V=800.0 PL=0
MOVL C01524 V=800.0 PL=0
MOVL C01525 V=800.0 PL=0
MOVL C01526 V=800.0 PL=0
MOVL C01527 V=800.0 PL=0
MOVL C01528 V=800.0 PL=0
MOVL C01529 V=800.0 PL=0
MOVL C01530 V=800.0 PL=0
MOVL C01531 V=800.0 PL=0
MOVL C01532 V=800.0 PL=0
MOVL C01533 V=800.0 PL=0
MOVL C01534 V=800.0 PL=0
MOVL C01535 V=800.0 PL=0
MOVL C01536 V=800.0 PL=0
MOVL C01537 V=800.0 PL=0
MOVL C01538 V=800.0 PL=0
MOVL C01539 V=800.0 PL=0
MOVL C01540 V=800.0 PL=0
MOVL C01541 V=800.0 PL=0
MOVL C01542 V=800.0 PL=0
MOVL C01543 V=800.0 PL=0
MOVL C01544 V=800.0 PL=0
MOVL C01545 V=800.0 PL=0
MOVL C01546 V=800.0 PL=0
MOVL C01547 V=800.0 PL=0
MOVL C01548 V=800.0 PL=0
MOVL C01549 V=800.0 PL=0
MOVL C01550 V=800.0 PL=0
MOVL C01551 V=800.0 PL=0
MOVL C01552 V=800.0 PL=0
MOVL C01553 V=800.0 PL=0
MOVL C01554 V=800.0 PL=0
MOVL C01555 V=800.0 PL=0
MOVL C01556 V=800.0 PL=0
MOVL C01557 V=800.0 PL=0
MOVL C01558 V=800.0 PL=0
MOVL C01559 V=800.0 PL=0
MOVL C01560 V=800.0 PL=0
MOVL C01561 V=800.0 PL=0
MOVL C01562 V=800.0 PL=0
MOVL C01563 V=800.0 PL=0
MOVL C01564 V=800.0 PL=0
MOVL C01565 V=800.0 PL=0
MOVL C01566 V=800.0 PL=0
MOVL C01567 V=800.0 PL=0
MOVL C01568 V=800.0 PL=0
MOVL C01569 V=800.0 PL=0
MOVL C01570 V=800.0 PL=0
MOVL C01571 V=800.0 PL=0
MOVL C01572 V=800.0 PL=0
MOVL C01573 V=800.0 PL=0
MOVL C01574 V=800.0 PL=0
MOVL C01575 V=800.0 PL=0
MOVL C01576 V=800.0 PL=0
MOVL C01577 V=800.0 PL=0
MOVL C01578 V=800.0 PL=0
MOVL C01579 V=800.0 PL=0
MOVL C01580 V=800.0 PL=0
MOVL C01581 V=800.0 PL=0
MOVL C01582 V=800.0 PL=0
MOVL C01583 V=800.0 PL=0
MOVL C01584 V=800.0 PL=0
MOVL C01585 V=800.0 PL=0
MOVL C01586 V=800.0 PL=0
MOVL C01587 V=800.0 PL=0
MOVL C01588 V=800.0 PL=0
MOVL C01589 V=800.0 PL=0
MOVL C01590 V=800.0 PL=0
MOVL C01591 V=800.0 PL=0
MOVL C01592 V=800.0 PL=0
MOVL C01593 V=800.0 PL=0
MOVL C01594 V=800.0 PL=0
MOVL C01595 V=800.0 PL=0
MOVL C01596 V=800.0 PL=0
MOVL C01597 V=800.0 PL=0
MOVL C01598 V=800.0 PL=0
MOVL C01599 V=800.0 PL=0
MOVL C01600 V=800.0 PL=0
MOVL C01601 V=800.0 PL=0
MOVL C01602 V=800.0 PL=0
MOVL C01603 V=800.0 PL=0
MOVL C01604 V=800.0 PL=0
MOVL C01605 V=800.0 PL=0
MOVL C01606 V=800.0 PL=0
MOVL C01607 V=800.0 PL=0
MOVL C01608 V=800.0 PL=0
MOVL C01609 V=800.0 PL=0
MOVL C01610 V=800.0 PL=0
MOVL C01611 V=800.0 PL=0
MOVL C01612 V=800.0 PL=0
MOVL C01613 V=800.0 PL=0
MOVL C01614 V=800.0 PL=0
MOVL C01615 V=800.0 PL=0
MOVL C01616 V=800.0 PL=0
MOVL C01617 V=800.0 PL=0
MOVL C01618 V=800.0 PL=0
MOVL C01619 V=800.0 PL=0
MOVL C01620 V=800.0 PL=0
MOVL C01621 V=800.0 PL=0
MOVL C01622 V=800.0 PL=0
MOVL C01623 V=800.0 PL=0
MOVL C01624 V=800.0 PL=0
MOVL C01625 V=800.0 PL=0
MOVL C01626 V=800.0 PL=0
MOVL C01627 V=800.0 PL=0
MOVL C01628 V=800.0 PL=0
MOVL C01629 V=800.0 PL=0
MOVL C01630 V=800.0 PL=0
MOVL C01631 V=800.0 PL=0
MOVL C01632 V=800.0 PL=0
MOVL C01633 V=800.0 PL=0
MOVL C01634 V=800.0 PL=0
MOVL C01635 V=800.0 PL=0
MOVL C01636 V=800.0 PL=0
MOVL C01637 V=800.0 PL=0
MOVL C01638 V=800.0 PL=0
MOVL C01639 V=800.0 PL=0
MOVL C01640 V=800.0 PL=0
MOVL C01641 V=800.0 PL=0
MOVL C01642 V=800.0 PL=0
MOVL C01643 V=800.0 PL=0
MOVL C01644 V=800.0 PL=0
MOVL C01645 V=800.0 PL=0
MOVL C01646 V=800.0 PL=0
MOVL C01647 V=800.0 PL=0
MOVL C01648 V=800.0 PL=0
MOVL C01649 V=800.0 PL=0
MOVL C01650 V=800.0 PL=0
MOVL C01651 V=800.0 PL=0
MOVL C01652 V=800.0 PL=0
MOVL C01653 V=800.0 PL=0
MOVL C01654 V=800.0 PL=0
MOVL C01655 V=800.0 PL=0
MOVL C01656 V=800.0 PL=0
MOVL C01657 V=800.0 PL=0
MOVL C01658 V=800.0 PL=0
MOVL C01659 V=800.0 PL=0
MOVL C01660 V=800.0 PL=0
MOVL C01661 V=800.0 PL=0
MOVL C01662 V=800.0 PL=0
MOVL C01663 V=800.0 PL=0
MOVL C01664 V=800.0 PL=0
MOVL C01665 V=800.0 PL=0
MOVL C01666 V=800.0 PL=0
MOVL C01667 V=800.0 PL=0
MOVL C01668 V=800.0 PL=0
MOVL C01669 V=800.0 PL=0
MOVL C01670 V=800.0 PL=0
MOVL C01671 V=800.0 PL=0
MOVL C01672 V=800.0 PL=0
MOVL C01673 V=800.0 PL=0
MOVL C01674 V=800.0 PL=0
MOVL C01675 V=800.0 PL=0
MOVL C01676 V=800.0 PL=0
MOVL C01677 V=800.0 PL=0
MOVL C01678 V=800.0 PL=0
MOVL C01679 V=800.0 PL=0
MOVL C01680 V=800.0 PL=0
MOVL C01681 V=800.0 PL=0
MOVL C01682 V=800.0 PL=0
MOVL C01683 V=800.0 PL=0
MOVL C01684 V=800.0 PL=0
MOVL C01685 V=800.0 PL=0
MOVL C01686 V=800.0 PL=0
MOVL C01687 V=800.0 PL=0
MOVL C01688 V=800.0 PL=0
MOVL C01689 V=800.0 PL=0
MOVL C01690 V=800.0 PL=0
MOVL C01691 V=800.0 PL=0
MOVL C01692 V=800.0 PL=0
MOVL C01693 V=800.0 PL=0
MOVL C01694 V=800.0 PL=0
MOVL C01695 V=800.0 PL=0
MOVL C01696 V=800.0 PL=0
MOVL C01697 V=800.0 PL=0
MOVL C01698 V=800.0 PL=0
MOVL C01699 V=800.0 PL=0
MOVL C01700 V=800.0 PL=0
MOVL C01701 V=800.0 PL=0
MOVL C01702 V=800.0 PL=0
MOVL C01703 V=800.0 PL=0
MOVL C01704 V=800.0 PL=0
MOVL C01705 V=800.0 PL=0
MOVL C01706 V=800.0 PL=0
MOVL C01707 V=800.0 PL=0
MOVL C01708 V=800.0 PL=0
MOVL C01709 V=800.0 PL=0
MOVL C01710 V=800.0 PL=0
MOVL C01711 V=800.0 PL=0
MOVL C01712 V=800.0 PL=0
MOVL C01713 V=800.0 PL=0
MOVL C01714 V=800.0 PL=0
MOVL C01715 V=800.0 PL=0
MOVL C01716 V=800.0 PL=0
MOVL C01717 V=800.0 PL=0
MOVL C01718 V=800.0 PL=0
MOVL C01719 V=800.0 PL=0
MOVL C01720 V=800.0 PL=0
MOVL C01721 V=800.0 PL=0
MOVL C01722 V=800.0 PL=0
MOVL C01723 V=800.0 PL=0
MOVL C01724 V=800.0 PL=0
MOVL C01725 V=800.0 PL=0
MOVL C01726 V=800.0 PL=0
MOVL C01727 V=800.0 PL=0
MOVL C01728 V=800.0 PL=0
MOVL C01729 V=800.0 PL=0
MOVL C01730 V=800.0 PL=0
MOVL C01731 V=800.0 PL=0
MOVL C01732 V=800.0 PL=0
MOVL C01733 V=800.0 PL=0
MOVL C01734 V=800.0 PL=0
MOVL C01735 V=800.0 PL=0
MOVL C01736 V=800.0 PL=0
MOVL C01737 V=800.0 PL=0
MOVL C01738 V=800.0 PL=0
MOVL C01739 V=800.0 PL=0
MOVL C01740 V=800.0 PL=0
MOVL C01741 V=800.0 PL=0
MOVL C01742 V=800.0 PL=0
MOVL C01743 V=800.0 PL=0
MOVL C01744 V=800.0 PL=0
MOVL C01745 V=800.0 PL=0
MOVL C01746 V=800.0 PL=0
MOVL C01747 V=800.0 PL=0
MOVL C01748 V=800.0 PL=0
MOVL C01749 V=800.0 PL=0
MOVL C01750 V=800.0 PL=0
MOVL C01751 V=800.0 PL=0
MOVL C01752 V=800.0 PL=0
MOVL C01753 V=800.0 PL=0
MOVL C01754 V=800.0 PL=0
MOVL C01755 V=800.0 PL=0
MOVL C01756 V=800.0 PL=0
MOVL C01757 V=800.0 PL=0
MOVL C01758 V=800.0 PL=0
MOVL C01759 V=800.0 PL=0
MOVL C01760 V=800.0 PL=0
MOVL C01761 V=800.0 PL=0
MOVL C01762 V=800.0 PL=0
MOVL C01763 V=800.0 PL=0
MOVL C01764 V=800.0 PL=0
MOVL C01765 V=800.0 PL=0
MOVL C01766 V=800.0 PL=0
MOVL C01767 V=800.0 PL=0
MOVL C01768 V=800.0 PL=0
MOVL C01769 V=800.0 PL=0
MOVL C01770 V=800.0 PL=0
MOVL C01771 V=800.0 PL=0
MOVL C01772 V=800.0 PL=0
MOVL C01773 V=800.0 PL=0
MOVL C01774 V=800.0 PL=0
MOVL C01775 V=800.0 PL=0
MOVL C01776 V=800.0 PL=0
MOVL C01777 V=800.0 PL=0
MOVL C01778 V=800.0 PL=0
MOVL C01779 V=800.0 PL=0
MOVL C01780 V=800.0 PL=0
MOVL C01781 V=800.0 PL=0
MOVL C01782 V=800.0 PL=0
MOVL C01783 V=800.0 PL=0
MOVL C01784 V=800.0 PL=0
MOVL C01785 V=800.0 PL=0
MOVL C01786 V=800.0 PL=0
MOVL C01787 V=800.0 PL=0
MOVL C01788 V=800.0 PL=0
MOVL C01789 V=800.0 PL=0
MOVL C01790 V=800.0 PL=0
MOVL C01791 V=800.0 PL=0
MOVL C01792 V=800.0 PL=0
MOVL C01793 V=800.0 PL=0
MOVL C01794 V=800.0 PL=0
MOVL C01795 V=800.0 PL=0
MOVL C01796 V=800.0 PL=0
MOVL C01797 V=800.0 PL=0
MOVL C01798 V=800.0 PL=0
MOVL C01799 V=800.0 PL=0
MOVL C01800 V=800.0 PL=0
MOVL C01801 V=800.0 PL=0
MOVL C01802 V=800.0 PL=0
MOVL C01803 V=800.0 PL=0
MOVL C01804 V=800.0 PL=0
MOVL C01805 V=800.0 PL=0
MOVL C01806 V=800.0 PL=0
MOVL C01807 V=800.0 PL=0
MOVL C01808 V=800.0 PL=0
MOVL C01809 V=800.0 PL=0
MOVL C01810 V=800.0 PL=0
MOVL C01811 V=800.0 PL=0
MOVL C01812 V=800.0 PL=0
MOVL C01813 V=800.0 PL=0
MOVL C01814 V=800.0 PL=0
MOVL C01815 V=800.0 PL=0
MOVL C01816 V=800.0 PL=0
MOVL C01817 V=800.0 PL=0
MOVL C01818 V=800.0 PL=0
MOVL C01819 V=800.0 PL=0
MOVL C01820 V=800.0 PL=0
MOVL C01821 V=800.0 PL=0
MOVL C01822 V=800.0 PL=0
MOVL C01823 V=800.0 PL=0
MOVL C01824 V=800.0 PL=0
MOVL C01825 V=800.0 PL=0
MOVL C01826 V=800.0 PL=0
MOVL C01827 V=800.0 PL=0
MOVL C01828 V=800.0 PL=0
MOVL C01829 V=800.0 PL=0
MOVL C01830 V=800.0 PL=0
MOVL C01831 V=800.0 PL=0
MOVL C01832 V=800.0 PL=0
MOVL C01833 V=800.0 PL=0
MOVL C01834 V=800.0 PL=0
MOVL C01835 V=800.0 PL=0
MOVL C01836 V=800.0 PL=0
MOVL C01837 V=800.0 PL=0
MOVL C01838 V=800.0 PL=0
MOVL C01839 V=800.0 PL=0
MOVL C01840 V=800.0 PL=0
MOVL C01841 V=800.0 PL=0
MOVL C01842 V=800.0 PL=0
MOVL C01843 V=800.0 PL=0
MOVL C01844 V=800.0 PL=0
MOVL C01845 V=800.0 PL=0
MOVL C01846 V=800.0 PL=0
MOVL C01847 V=800.0 PL=0
MOVL C01848 V=800.0 PL=0
MOVL C01849 V=800.0 PL=0
MOVL C01850 V=800.0 PL=0
MOVL C01851 V=800.0 PL=0
MOVL C01852 V=800.0 PL=0
MOVL C01853 V=800.0 PL=0
MOVL C01854 V=800.0 PL=0
MOVL C01855 V=800.0 PL=0
MOVL C01856 V=800.0 PL=0
MOVL C01857 V=800.0 PL=0
MOVL C01858 V=800.0 PL=0
MOVL C01859 V=800.0 PL=0
MOVL C01860 V=800.0 PL=0
MOVL C01861 V=800.0 PL=0
MOVL C01862 V=800.0 PL=0
MOVL C01863 V=800.0 PL=0
MOVL C01864 V=800.0 PL=0
MOVL C01865 V=800.0 PL=0
MOVL C01866 V=800.0 PL=0
MOVL C01867 V=800.0 PL=0
MOVL C01868 V=800.0 PL=0
MOVL C01869 V=800.0 PL=0
MOVL C01870 V=800.0 PL=0
MOVL C01871 V=800.0 PL=0
MOVL C01872 V=800.0 PL=0
MOVL C01873 V=800.0 PL=0
MOVL C01874 V=800.0 PL=0
MOVL C01875 V=800.0 PL=0
MOVL C01876 V=800.0 PL=0
MOVL C01877 V=800.0 PL=0
MOVL C01878 V=800.0 PL=0
MOVL C01879 V=800.0 PL=0
MOVL C01880 V=800.0 PL=0
MOVL C01881 V=800.0 PL=0
MOVL C01882 V=800.0 PL=0
MOVL C01883 V=800.0 PL=0
MOVL C01884 V=800.0 PL=0
MOVL C01885 V=800.0 PL=0
MOVL C01886 V=800.0 PL=0
MOVL C01887 V=800.0 PL=0
MOVL C01888 V=800.0 PL=0
MOVL C01889 V=800.0 PL=0
MOVL C01890 V=800.0 PL=0
MOVL C01891 V=800.0 PL=0
MOVL C01892 V=800.0 PL=0
MOVL C01893 V=800.0 PL=0
MOVL C01894 V=800.0 PL=0
MOVL C01895 V=800.0 PL=0
MOVL C01896 V=800.0 PL=0
MOVL C01897 V=800.0 PL=0
MOVL C01898 V=800.0 PL=0
MOVL C01899 V=800.0 PL=0
MOVL C01900 V=800.0 PL=0
MOVL C01901 V=800.0 PL=0
MOVL C01902 V=800.0 PL=0
MOVL C01903 V=800.0 PL=0
MOVL C01904 V=800.0 PL=0
MOVL C01905 V=800.0 PL=0
MOVL C01906 V=800.0 PL=0
MOVL C01907 V=800.0 PL=0
MOVL C01908 V=800.0 PL=0
MOVL C01909 V=800.0 PL=0
MOVL C01910 V=800.0 PL=0
MOVL C01911 V=800.0 PL=0
MOVL C01912 V=800.0 PL=0
MOVL C01913 V=800.0 PL=0
MOVL C01914 V=800.0 PL=0
MOVL C01915 V=800.0 PL=0
MOVL C01916 V=800.0 PL=0
MOVL C01917 V=800.0 PL=0
MOVL C01918 V=800.0 PL=0
MOVL C01919 V=800.0 PL=0
MOVL C01920 V=800.0 PL=0
MOVL C01921 V=800.0 PL=0
MOVL C01922 V=800.0 PL=0
MOVL C01923 V=800.0 PL=0
MOVL C01924 V=800.0 PL=0
MOVL C01925 V=800.0 PL=0
MOVL C01926 V=800.0 PL=0
MOVL C01927 V=800.0 PL=0
MOVL C01928 V=800.0 PL=0
MOVL C01929 V=800.0 PL=0
MOVL C01930 V=800.0 PL=0
MOVL C01931 V=800.0 PL=0
MOVL C01932 V=800.0 PL=0
MOVL C01933 V=800.0 PL=0
MOVL C01934 V=800.0 PL=0
MOVL C01935 V=800.0 PL=0
MOVL C01936 V=800.0 PL=0
MOVL C01937 V=800.0 PL=0
MOVL C01938 V=800.0 PL=0
MOVL C01939 V=800.0 PL=0
MOVL C01940 V=800.0 PL=0
MOVL C01941 V=800.0 PL=0
MOVL C01942 V=800.0 PL=0
MOVL C01943 V=800.0 PL=0
MOVL C01944 V=800.0 PL=0
MOVL C01945 V=800.0 PL=0
MOVL C01946 V=800.0 PL=0
MOVL C01947 V=800.0 PL=0
MOVL C01948 V=800.0 PL=0
MOVL C01949 V=800.0 PL=0
MOVL C01950 V=800.0 PL=0
MOVL C01951 V=800.0 PL=0
MOVL C01952 V=800.0 PL=0
MOVL C01953 V=800.0 PL=0
MOVL C01954 V=800.0 PL=0
MOVL C01955 V=800.0 PL=0
MOVL C01956 V=800.0 PL=0
MOVL C01957 V=800.0 PL=0
MOVL C01958 V=800.0 PL=0
MOVL C01959 V=800.0 PL=0
MOVL C01960 V=800.0 PL=0
MOVL C01961 V=800.0 PL=0
MOVL C01962 V=800.0 PL=0
MOVL C01963 V=800.0 PL=0
MOVL C01964 V=800.0 PL=0
MOVL C01965 V=800.0 PL=0
MOVL C01966 V=800.0 PL=0
MOVL C01967 V=800.0 PL=0
MOVL C01968 V=800.0 PL=0
MOVL C01969 V=800.0 PL=0
MOVL C01970 V=800.0 PL=0
MOVL C01971 V=800.0 PL=0
MOVL C01972 V=800.0 PL=0
MOVL C01973 V=800.0 PL=0
MOVL C01974 V=800.0 PL=0
MOVL C01975 V=800.0 PL=0
MOVL C01976 V=800.0 PL=0
MOVL C01977 V=800.0 PL=0
MOVL C01978 V=800.0 PL=0
MOVL C01979 V=800.0 PL=0
MOVL C01980 V=800.0 PL=0
MOVL C01981 V=800.0 PL=0
MOVL C01982 V=800.0 PL=0
MOVL C01983 V=800.0 PL=0
MOVL C01984 V=800.0 PL=0
MOVL C01985 V=800.0 PL=0
MOVL C01986 V=800.0 PL=0
MOVL C01987 V=800.0 PL=0
MOVL C01988 V=800.0 PL=0
MOVL C01989 V=800.0 PL=0
MOVL C01990 V=800.0 PL=0
MOVL C01991 V=800.0 PL=0
MOVL C01992 V=800.0 PL=0
MOVL C01993 V=800.0 PL=0
MOVL C01994 V=800.0 PL=0
MOVL C01995 V=800.0 PL=0
MOVL C01996 V=800.0 PL=0
MOVL C01997 V=800.0 PL=0
MOVL C01998 V=800.0 PL=0
MOVL C01999 V=800.0 PL=0
MOVL C02000 V=800.0 PL=0
MOVL C02001 V=800.0 PL=0
MOVL C02002 V=800.0 PL=0
MOVL C02003 V=800.0 PL=0
MOVL C02004 V=800.0 PL=0
MOVL C02005 V=800.0 PL=0
MOVL C02006 V=800.0 PL=0
MOVL C02007 V=800.0 PL=0
MOVL C02008 V=800.0 PL=0
MOVL C02009 V=800.0 PL=0
MOVL C02010 V=800.0 PL=0
MOVL C02011 V=800.0 PL=0
MOVL C02012 V=800.0 PL=0
MOVL C02013 V=800.0 PL=0
MOVL C02014 V=800.0 PL=0
MOVL C02015 V=800.0 PL=0
MOVL C02016 V=800.0 PL=0
MOVL C02017 V=800.0 PL=0
MOVL C02018 V=800.0 PL=0
MOVL C02019 V=800.0 PL=0
MOVL C02020 V=800.0 PL=0
MOVL C02021 V=800.0 PL=0
MOVL C02022 V=800.0 PL=0
MOVL C02023 V=800.0 PL=0
MOVL C02024 V=800.0 PL=0
MOVL C02025 V=800.0 PL=0
MOVL C02026 V=800.0 PL=0
MOVL C02027 V=800.0 PL=0
MOVL C02028 V=800.0 PL=0
MOVL C02029 V=800.0 PL=0
MOVL C02030 V=800.0 PL=0
MOVL C02031 V=800.0 PL=0
MOVL C02032 V=800.0 PL=0
MOVL C02033 V=800.0 PL=0
MOVL C02034 V=800.0 PL=0
MOVL C02035 V=800.0 PL=0
MOVL C02036 V=800.0 PL=0
MOVL C02037 V=800.0 PL=0
MOVL C02038 V=800.0 PL=0
MOVL C02039 V=800.0 PL=0
MOVL C02040 V=800.0 PL=0
MOVL C02041 V=800.0 PL=0
MOVL C02042 V=800.0 PL=0
MOVL C02043 V=800.0 PL=0
MOVL C02044 V=800.0 PL=0
MOVL C02045 V=800.0 PL=0
MOVL C02046 V=800.0 PL=0
MOVL C02047 V=800.0 PL=0
MOVL C02048 V=800.0 PL=0
MOVL C02049 V=800.0 PL=0
MOVL C02050 V=800.0 PL=0
MOVL C02051 V=800.0 PL=0
MOVL C02052 V=800.0 PL=0
MOVL C02053 V=800.0 PL=0
MOVL C02054 V=800.0 PL=0
MOVL C02055 V=800.0 PL=0
MOVL C02056 V=800.0 PL=0
MOVL C02057 V=800.0 PL=0
MOVL C02058 V=800.0 PL=0
MOVL C02059 V=800.0 PL=0
MOVL C02060 V=800.0 PL=0
MOVL C02061 V=800.0 PL=0
MOVL C02062 V=800.0 PL=0
MOVL C02063 V=800.0 PL=0
MOVL C02064 V=800.0 PL=0
MOVL C02065 V=800.0 PL=0
MOVL C02066 V=800.0 PL=0
MOVL C02067 V=800.0 PL=0
MOVL C02068 V=800.0 PL=0
MOVL C02069 V=800.0 PL=0
MOVL C02070 V=800.0 PL=0
MOVL C02071 V=800.0 PL=0
MOVL C02072 V=800.0 PL=0
MOVL C02073 V=800.0 PL=0
MOVL C02074 V=800.0 PL=0
MOVL C02075 V=800.0 PL=0
MOVL C02076 V=800.0 PL=0
MOVL C02077 V=800.0 PL=0
MOVL C02078 V=800.0 PL=0
MOVL C02079 V=800.0 PL=0
MOVL C02080 V=800.0 PL=0
MOVL C02081 V=800.0 PL=0
MOVL C02082 V=800.0 PL=0
MOVL C02083 V=800.0 PL=0
MOVL C02084 V=800.0 PL=0
MOVL C02085 V=800.0 PL=0
MOVL C02086 V=800.0 PL=0
MOVL C02087 V=800.0 PL=0
MOVL C02088 V=800.0 PL=0
MOVL C02089 V=800.0 PL=0
MOVL C02090 V=800.0 PL=0
MOVL C02091 V=800.0 PL=0
MOVL C02092 V=800.0 PL=0
MOVL C02093 V=800.0 PL=0
MOVL C02094 V=800.0 PL=0
MOVL C02095 V=800.0 PL=0
MOVL C02096 V=800.0 PL=0
MOVL C02097 V=800.0 PL=0
MOVL C02098 V=800.0 PL=0
MOVL C02099 V=800.0 PL=0
MOVL C02100 V=800.0 PL=0
MOVL C02101 V=800.0 PL=0
MOVL C02102 V=800.0 PL=0
MOVL C02103 V=800.0 PL=0
MOVL C02104 V=800.0 PL=0
MOVL C02105 V=800.0 PL=0
MOVL C02106 V=800.0 PL=0
MOVL C02107 V=800.0 PL=0
MOVL C02108 V=800.0 PL=0
MOVL C02109 V=800.0 PL=0
MOVL C02110 V=800.0 PL=0
MOVL C02111 V=800.0 PL=0
MOVL C02112 V=800.0 PL=0
MOVL C02113 V=800.0 PL=0
MOVL C02114 V=800.0 PL=0
MOVL C02115 V=800.0 PL=0
MOVL C02116 V=800.0 PL=0
MOVL C02117 V=800.0 PL=0
MOVL C02118 V=800.0 PL=0
MOVL C02119 V=800.0 PL=0
MOVL C02120 V=800.0 PL=0
MOVL C02121 V=800.0 PL=0
MOVL C02122 V=800.0 PL=0
MOVL C02123 V=800.0 PL=0
MOVL C02124 V=800.0 PL=0
MOVL C02125 V=800.0 PL=0
MOVL C02126 V=800.0 PL=0
MOVL C02127 V=800.0 PL=0
MOVL C02128 V=800.0 PL=0
MOVL C02129 V=800.0 PL=0
MOVL C02130 V=800.0 PL=0
MOVL C02131 V=800.0 PL=0
MOVL C02132 V=800.0 PL=0
